		;
		// evtl. wait time if reset of device is necessary and then decide to go to states or ERROR state
		IF (CIf.Job.bolAlmReset = TRUE) THEN
			CIf.Job.eMe_ActivAlmClass := E_AlmClass.NONE; // reset feedback channel for parent
			CIf.Job.bolAlmReset := FALSE;
		END_IF
		// **************************************************************************
		// Wait until Reset all CRC Error is Done
		// **************************************************************************
			fbEcMasterFrameStatisticClearCRC(bExecute:= FALSE);
			// Wait until done
			IF NOT (fbEcMasterFrameStatisticClearCRC.bBusy) THEN
				IF NOT (fbEcMasterFrameStatisticClearCRC.bError) THEN
					bolResetCRCError := FALSE;
				// Error
				ELSE
					// SIf.Alm[E_ALM_ECD.ADS_ComError].strText := 'ADS Communication Error to EtherCAT Master'; // ADS Communication Error to EtherCAT Master => Info = ADS_Errorcode
					pfbAlarmCtrl^.setAlarm(CIf.Info.intCtrlId,E_ALM_ECD.ADS_ComError,UDINT_TO_DINT(fbEcGetSlaveCrcError.nErrId),ADR(SIf.Alm),E_AlmState.RST,CIf.Job.eMe_ActivAlmClass);
					me.StateMachine.intStateNext := cSTA_SUB_ERROR;		
				END_IF
			END_IF
		
		// State Change Condition
		IF ((CIf.Job.bolAlmReset = FALSE) AND (bolResetCRCError = FALSE)) THEN
			IF (me.StateMachine.intStateHistory<=cSTA_PON) THEN
				me.StateMachine.intStateNext := cSTA_PONBusy;
			ELSIF ((SIf.Cfg.bolRunAlways = TRUE) OR (me.intCmd=BASE_PLC.cCMD_RUN)) THEN
				me.StateMachine.intStateNext := cSTA_RUNBusy;
			ELSE
				me.StateMachine.intStateNext := cSTA_OFFBusy;
			END_IF
		END_IF
	END_IF


//--------------------------------------------------------------------------------------
// Exit action
	IF (me.StateMachine.intState<>me.StateMachine.intStateNext) THEN
		;
	END_IF
END_METHOD

METHOD PROTECTED sta_OFF : BOOL
// state implemetation
//--------------------------------------------------------------------------------------
// Entry action
	IF (me.StateMachine.intState<>me.StateMachine.intStateLastCycle) THEN
		me.StateMachine.intStateLastCycle := me.StateMachine.intState;
		// Initialize sub state machine
		me.SubStateMachine.intState:= cSTA_SUB_INITIALIZE; 
		me.SubStateMachine.intStateNext := cSTA_SUB_INITIALIZE;
	END_IF
	
//--------------------------------------------------------------------------------------
// Cyclic action
	IF (me.StateMachine.intState=me.StateMachine.intStateLastCycle) THEN	
		// State Change Condition
		IF (me.Alarm.eActivAlmClass<>E_AlmClass.EOFF) AND (me.Alarm.eActivAlmClass<>E_AlmClass.OFF) THEN	
			IF ((SIf.Cfg.bolRunAlways = TRUE) OR (me.intCmd=BASE_PLC.cCMD_RUN))  THEN
				me.StateMachine.intStateNext := BASE_PLC.cSTA_RUNBusy;
			END_IF
		END_IF
	END_IF

//--------------------------------------------------------------------------------------
// Exit action
	IF (me.StateMachine.intState<>me.StateMachine.intStateNext) THEN
		;
	END_IF
END_METHOD

METHOD PROTECTED sta_PON : BOOL
// state implemetation
//--------------------------------------------------------------------------------------
// Entry action
	IF (me.StateMachine.intState<>me.StateMachine.intStateLastCycle) THEN
		me.StateMachine.intStateLastCycle := me.StateMachine.intState;
		
	END_IF

//--------------------------------------------------------------------------------------
// Cyclic action
	IF (me.StateMachine.intState=me.StateMachine.intStateLastCycle) THEN
		
		;	
		// State Change Condition
		IF ((me.intCmd<>cCMD_PON) AND (me.intCmd<>cCMD_DONE)) OR (SIf.Cfg.bolRunAlways = TRUE) THEN
			me.StateMachine.intStateNext := BASE_PLC.cSTA_OFFBusy;
		END_IF
	END_IF

//--------------------------------------------------------------------------------------
// Exit action
	IF (me.StateMachine.intState<>me.StateMachine.intStateNext) THEN
		;
	END_IF
END_METHOD

METHOD PROTECTED sta_PONBusy : BOOL
VAR
	ii: UINT;
	/// Internal Variable for Found Address
	bolSlaveOK: BOOL;
END_VAR
// state implemetation
//--------------------------------------------------------------------------------------
// Entry action
	IF (me.StateMachine.intState<>me.StateMachine.intStateLastCycle) THEN
		me.StateMachine.intStateLastCycle := me.StateMachine.intState;
		
		udiNumOfStateErrors:= 0;
		udiNumOfCRCErrors:= 0;
		uinLoop:= 0;
		uinSlaveNbr:= 0;

		// Initialize sub state machine
		me.SubStateMachine.intState:= cSTA_SUB_INITIALIZE; 
		me.SubStateMachine.intStateNext := cSTA_SUB_INITIALIZE;
		
		// Get stored alarmtextes into local Texts
		FOR ii := 1 TO (E_ALM_ECD.MAX_E_ALM - 1) DO
			arrAlmtexts[ii] := SIf.Alm[ii].strText;
		END_FOR
	END_IF

//--------------------------------------------------------------------------------------
// Cyclic action
	IF (me.StateMachine.intState=me.StateMachine.intStateLastCycle) THEN
			// Simulation
			IF (CIf.SwCfg.bolSimulation) THEN
				me.SubStateMachine.intStateNext := cSTA_SUB_DONE;
			END_IF
		
			// Sub statemachine to set necessary AMS routes and determine the handle ID of all connections in list	
			CASE me.SubStateMachine.intState OF	
			
				cSTA_SUB_INITIALIZE: 
					me.SubStateMachine.intStateNext := cSTA_SUB_CheckMaster;		

				
				// **************************************************************************
				// Call FUB fbEcGetMasterState to get The State of the EtherCAT Master Device
				// **************************************************************************
				cSTA_SUB_CheckMaster:
				
					// Prepare Function Block
					fbEcGetMasterState(sNetId:= SIf.Cfg.strNetID, 
										bExecute:= FALSE, 
										tTimeout:= UDINT_TO_TIME(SIf.Par.udiTOCheckAll_ms)); 
				
					// Start Function
					fbEcGetMasterState(bExecute:= TRUE, 
										tTimeout:= UDINT_TO_TIME(SIf.Par.udiTOCheckAll_ms)); 
				
					me.SubStateMachine.intStateNext := cSTA_SUB_CheckMasterDone;		
							
				// **************************************************************************
				// Wait until GetAllSlaveAdress is Done
				// **************************************************************************
				cSTA_SUB_CheckMasterDone:
				
					fbEcGetMasterState(bExecute:= FALSE);
					// Wait until done
					IF NOT (fbEcGetMasterState.bBusy) THEN
						IF NOT (fbEcGetMasterState.bError) THEN
							SIf.Cur.worMasterState := fbEcGetMasterState.state;
							// In Operational State check slaves
							IF SIf.Cur.worMasterState = Tc2_EtherCAT.EC_DEVICE_STATE_OP THEN
								me.SubStateMachine.intStateNext := cSTA_SUB_GetAllSlaveAdress;
							// In Pre-Operational check again
							ELSIF ((SIf.Cur.worMasterState = Tc2_EtherCAT.EC_DEVICE_STATE_PREOP) OR (SIf.Cur.worMasterState = Tc2_EtherCAT.EC_DEVICE_STATE_PREOP)) THEN
								me.SubStateMachine.intStateNext := cSTA_SUB_CheckMaster;
							// ELSE ERROR
							ELSE
								// SIf.Alm[E_ALM_ECD.MasterStateError].strText := 'Master State Error'; // Master not in the correct state => Info = Masterstate
								pfbAlarmCtrl^.setAlarm(CIf.Info.intCtrlId,E_ALM_ECD.MasterStateError,WORD_TO_DINT(SIf.Cur.worMasterState),ADR(SIf.Alm),E_AlmState.RST,CIf.Job.eMe_ActivAlmClass);								
							END_IF
						// Error
						ELSE
							// SIf.Alm[E_ALM_ECD.ADS_ComError].strText := 'ADS Communication Error to EtherCAT Master'; // ADS Communication Error to EtherCAT Master => Info = ADS_Errorcode
							pfbAlarmCtrl^.setAlarm(CIf.Info.intCtrlId,E_ALM_ECD.ADS_ComError,UDINT_TO_DINT(fbEcGetMasterState.nErrId),ADR(SIf.Alm),E_AlmState.RST,CIf.Job.eMe_ActivAlmClass);
							me.SubStateMachine.intStateNext := cSTA_SUB_ERROR;		
						END_IF
					END_IF
							
				
				// **************************************************************************
				// Call FUB fbEcGetAllSlaveAddr to get all connected slaves. 
				// **************************************************************************
				cSTA_SUB_GetAllSlaveAdress:
				
					// Prepare Function Block
					fbEcGetAllSlaveAddr(sNetId:= SIf.Cfg.strNetID, 
										pAddrBuf:= ADR(arrSlaveAdress), 
										cbBufLen:= SIZEOF(arrSlaveAdress), 
										bExecute:= FALSE, 
										tTimeout:= UDINT_TO_TIME(SIf.Par.udiTOCheckAll_ms));
				
					// Start Function
					fbEcGetAllSlaveAddr(bExecute:= TRUE, 
										tTimeout:= UDINT_TO_TIME(SIf.Par.udiTOCheckAll_ms));
				
					me.SubStateMachine.intStateNext := cSTA_SUB_GetAllSlaveAdressDone;		
							
				// **************************************************************************
				// Wait until GetAllSlaveAdress is Done
				// **************************************************************************
				cSTA_SUB_GetAllSlaveAdressDone:
				
					fbEcGetAllSlaveAddr(bExecute:= FALSE);
					// Wait until done
					IF NOT (fbEcGetAllSlaveAddr.bBusy) THEN
						IF NOT (fbEcGetAllSlaveAddr.bError) THEN
							// Prepare data
							SIf.Cur.uinNumOfSlaves := fbEcGetAllSlaveAddr.nSlaves;
							IF SIf.Cur.uinNumOfSlaves > 0 THEN
								FOR uinLoop := 0 TO (SIf.Cur.uinNumOfSlaves-1) DO
									SIf.Cur.stSlaveData[uinLoop].uinAddress := arrSlaveAdress[uinLoop];
								END_FOR
							ELSE
								// SIf.Alm[E_ALM_ECD.NoSlaveFound].strText :=  'No Slave in Network'; 		// No EtherCAT Slave found in the network
								pfbAlarmCtrl^.setAlarm(CIf.Info.intCtrlId,E_ALM_ECD.NoSlaveFound,0,ADR(SIf.Alm),E_AlmState.RST,CIf.Job.eMe_ActivAlmClass);								
							END_IF
							me.SubStateMachine.intStateNext := cSTA_SUB_GetConfSlaves;
						// Error
						ELSE
							// SIf.Alm[E_ALM_ECD.ADS_ComError].strText := 'ADS Communication Error to EtherCAT Master'; // ADS Communication Error to EtherCAT Master => Info = ADS_Errorcode
							pfbAlarmCtrl^.setAlarm(CIf.Info.intCtrlId,E_ALM_ECD.ADS_ComError,UDINT_TO_DINT(fbEcGetAllSlaveAddr.nErrId),ADR(SIf.Alm),E_AlmState.RST,CIf.Job.eMe_ActivAlmClass);
							me.SubStateMachine.intStateNext := cSTA_SUB_ERROR;		
						END_IF
					END_IF
			
				// **************************************************************************
				// Call FUB fbEcGetConfSlaves to get all configurated slaves. 
				// **************************************************************************
				cSTA_SUB_GetConfSlaves:
				
					// Prepare Function Block
					fbEcGetConfSlaves(sNetId:= SIf.Cfg.strNetID, 
										pArrEcConfSlaveInfo:= ADR(arrSlaveConf), 
										cbBufLen:= SIZEOF(arrSlaveConf), 
										bExecute:= FALSE, 
										tTimeout:= UDINT_TO_TIME(SIf.Par.udiTOCheckAll_ms));
				
					// Start Function
					fbEcGetConfSlaves(bExecute:= TRUE, 
										tTimeout:= UDINT_TO_TIME(SIf.Par.udiTOCheckAll_ms));
				
					me.SubStateMachine.intStateNext := cSTA_SUB_GetConfSlavesDone;		
							
				// **************************************************************************
				// Wait until fbEcGetConfSlaves is Done
				// **************************************************************************
				cSTA_SUB_GetConfSlavesDone:
				
					fbEcGetConfSlaves(bExecute:= FALSE);
					// Wait until done
					IF NOT (fbEcGetConfSlaves.bBusy) THEN
						IF NOT (fbEcGetConfSlaves.bError) THEN
							// Prepare data
							uinConfigSlaveNbr := fbEcGetConfSlaves.nSlaves;
							IF uinConfigSlaveNbr > 0 THEN
								uinErrorSlaveAdr := 0;
								uinErrorSlaveNbr := 0;
								// Search if configurated Address if found in the hardware found Slaves
								// Loop throug the Configrated Arreay...
								FOR ii := 0 TO (uinConfigSlaveNbr-1) DO	
									bolSlaveOK := FALSE;				
									//...and search in the found addresses	
									FOR uinLoop := 0 TO (SIf.Cur.uinNumOfSlaves-1) DO
										IF (WORD_TO_UINT(arrSlaveConf[ii].nAddr) = SIf.Cur.stSlaveData[uinLoop].uinAddress) THEN // Adress of Configurated and found Slave is the same
											// Copy configuration Data in the CUR Structure
											SIf.Cur.stSlaveData[uinLoop].stConfigData := arrSlaveConf[ii];
											// This slave is done
											bolSlaveOK := TRUE;
											EXIT;
										END_IF
									END_FOR
									// If configurated Address is not found in the redaed Hardware addresses, get Address and increment number
									IF bolSlaveOK = FALSE THEN
										IF uinErrorSlaveAdr = 0 THEN // only write the first module in Error as information
											uinErrorSlaveAdr := WORD_TO_UINT(arrSlaveConf[ii].nAddr);
										END_IF
										uinErrorSlaveNbr := uinErrorSlaveNbr + 1;
									END_IF
								END_FOR
								// Error handling if minimal one configurated slave not found
								IF uinErrorSlaveNbr > 0 THEN 		// Minimal one false Slave
									// Get Error Information
									dinAlarmInfo := UDINT_TO_DINT(SHL(UINT_TO_UDINT(uinErrorSlaveNbr),16) OR uinErrorSlaveAdr);
									strAlarminfo := CONCAT( 'Slave Number: ' , UINT_TO_STRING(uinErrorSlaveAdr));
									strAlarminfo := CONCAT(strAlarminfo, ' of totally missings: ');
									strAlarminfo := CONCAT(strAlarminfo, UDINT_TO_STRING(uinErrorSlaveNbr));
									
									SIf.Alm[E_ALM_ECD.NotAllSlaveConnected].strText := CONCAT(arrAlmtexts[E_ALM_ECD.NotAllSlaveConnected], strAlarminfo);
									
									// SIf.Alm[E_ALM_ECD.NotAllSlaveConnected].strText := 'Configuration and actual differences';// // Configured and reached Slaves are not the same => Info Byte 0+1 = Slave Addres from last error Info Byte 2+3 = Numbers of error Slaves
									pfbAlarmCtrl^.setAlarm(CIf.Info.intCtrlId,E_ALM_ECD.NotAllSlaveConnected,dinAlarmInfo,ADR(SIf.Alm),E_AlmState.RST,CIf.Job.eMe_ActivAlmClass);																	
								END_IF
								// If more slaves hardware found as configurated also an error
								IF SIf.Cur.uinNumOfSlaves > uinConfigSlaveNbr THEN
									// Search if hardware Address which is not configurated
									// Loop throug the Hardware Arreay...
									FOR uinLoop := 0 TO (SIf.Cur.uinNumOfSlaves-1) DO	
										bolSlaveOK := FALSE;				
										//...and search in the configuration
										FOR ii := 0 TO (uinConfigSlaveNbr-1) DO										
											IF (WORD_TO_UINT(arrSlaveConf[ii].nAddr) = SIf.Cur.stSlaveData[uinLoop].uinAddress) THEN // Adress of Configurated and found Slave is the same
												// This slave is done
												bolSlaveOK := TRUE;
												EXIT;
											END_IF
										END_FOR
										// If configurated Address is not found, get Address and increment number
										IF bolSlaveOK = FALSE THEN
											IF uinErrorSlaveAdr = 0 THEN // only write the first module in Error as information
												uinErrorSlaveAdr := WORD_TO_UINT(arrSlaveConf[ii].nAddr);
											END_IF
											uinErrorSlaveNbr := uinErrorSlaveNbr + 1;
										END_IF
									END_FOR
										// Error handling if minimal one configurated slave not found
										IF uinErrorSlaveNbr > 0 THEN 		// Minimal one false Slave
											// Get Error Information
											strAlarminfo := CONCAT(' Slave Number: ' , UINT_TO_STRING(uinErrorSlaveAdr));
											strAlarminfo := CONCAT(strAlarminfo, ' of totally missings: ');
											strAlarminfo := CONCAT(strAlarminfo, UDINT_TO_STRING(uinErrorSlaveNbr));
											
											SIf.Alm[E_ALM_ECD.ToManySlaves].strText := CONCAT(arrAlmtexts[E_ALM_ECD.ToManySlaves], strAlarminfo);
											dinAlarmInfo := UDINT_TO_DINT(SHL(UINT_TO_UDINT(uinErrorSlaveNbr),16) OR uinErrorSlaveAdr);
											// SIf.Alm[E_ALM_ECD.ToManySlaves].strText := 'To many slaves';// More slaves at the master as the structure could handle => Info Byte 0+1 = Slave Addres from last error Info Byte 2+3 = Numbers of error Slaves
											pfbAlarmCtrl^.setAlarm(CIf.Info.intCtrlId,E_ALM_ECD.ToManySlaves,dinAlarmInfo,ADR(SIf.Alm),E_AlmState.RST,CIf.Job.eMe_ActivAlmClass);																	
										END_IF										
								END_IF
							// No Slaves in Cofiguration Found	
							ELSE
								// SIf.Alm[E_ALM_ECD.NoSlaveFound].strText :=  'No Slave in Network'; 		// No EtherCAT Slave found in the network
								pfbAlarmCtrl^.setAlarm(CIf.Info.intCtrlId,E_ALM_ECD.NoSlaveFound,0,ADR(SIf.Alm),E_AlmState.RST,CIf.Job.eMe_ActivAlmClass);								
							END_IF
							me.SubStateMachine.intStateNext := cSTA_SUB_DONE;
						// Error
						ELSE
							// SIf.Alm[E_ALM_ECD.ADS_ComError].strText := 'ADS Communication Error to EtherCAT Master'; // ADS Communication Error to EtherCAT Master => Info = ADS_Errorcode
							pfbAlarmCtrl^.setAlarm(CIf.Info.intCtrlId,E_ALM_ECD.ADS_ComError,UDINT_TO_DINT(fbEcGetConfSlaves.nErrorId),ADR(SIf.Alm),E_AlmState.RST,CIf.Job.eMe_ActivAlmClass);
							me.SubStateMachine.intStateNext := cSTA_SUB_ERROR;		
						END_IF
					END_IF
			

				
				// **************************************************************************
				// All necessary AMS routes set and connection handles are determined 
				// **************************************************************************
				cSTA_SUB_DONE:
				
				// **************************************************************************
				// Error
				// **************************************************************************
				cSTA_SUB_ERROR:
				
			END_CASE	
			
		
		// State Change Condition
		IF ((me.SubStateMachine.intState=cSTA_SUB_ERROR) OR (me.StateMachine.udiTimeInState_ms >= SIf.Par.udiTOPowerOn_ms)) THEN
			// In case if TO
			IF (me.StateMachine.udiTimeInState_ms >= SIf.Par.udiTOPowerOn_ms) THEN
				// SIf.Alm[E_ALM_ECD.TimeOutFunction].strText := 'Timeout EtherCAT function'; // A Function is not finished after the defined Timeout
				pfbAlarmCtrl^.setAlarm(CIf.Info.intCtrlId,E_ALM_ECD.TimeOutFunction,UDINT_TO_DINT(me.StateMachine.udiTimeInState_ms),ADR(SIf.Alm),E_AlmState.RST,CIf.Job.eMe_ActivAlmClass);
			END_IF
			me.StateMachine.intStateNext := cSTA_ERROR;				
		ELSIF (me.SubStateMachine.intState=cSTA_SUB_DONE) THEN
			me.StateMachine.intStateNext := cSTA_PON;
		END_IF
			
	END_IF

//--------------------------------------------------------------------------------------
// Exit action
	IF (me.StateMachine.intState<>me.StateMachine.intStateNext) THEN
		;
	END_IF
END_METHOD

METHOD PROTECTED sta_RUN : BOOL
VAR
	/// internal Loop Variable
	intI: INT;
	/// Internal Variable for Found Address
	bolAlaveOK: BOOL;
END_VAR
// state implemetation
//--------------------------------------------------------------------------------------
// Entry action
	IF (me.StateMachine.intState<>me.StateMachine.intStateLastCycle) THEN
		me.StateMachine.intStateLastCycle := me.StateMachine.intState;
		
		udiNumOfStateErrors:= 0;
		udiNumOfCRCErrors:= 0;
		uinLoop:= 0;
		uinSlaveNbr:= 0;

		// Initialize sub state machine
		me.SubStateMachine.intState:= cSTA_SUB_INITIALIZE; 
		me.SubStateMachine.intStateNext := cSTA_SUB_INITIALIZE;
		
	END_IF

//--------------------------------------------------------------------------------------
// Cyclic action
	IF (me.StateMachine.intState=me.StateMachine.intStateLastCycle) THEN
			// Simulation
			IF (CIf.SwCfg.bolSimulation) THEN
				me.SubStateMachine.intStateNext := cSTA_SUB_WAIT_NEXT_POLL;
				me.SubStateMachine.udiTimeInState_ms := 0;
			END_IF
			
			// Check if a Reset of the CRC Errors has to be done
			IF ((SIf.Alm[E_ALM_ECD.SlaveCRCError].bol = TRUE) AND (CIf.Job.bolAlmReset = TRUE)) THEN
				bolResetCRCError := TRUE;
				SIf.Alm[E_ALM_ECD.SlaveCRCError].bol := FALSE;
			END_IF
			
		
			// Sub statemachine to set necessary AMS routes and determine the handle ID of all connections in list	
			CASE me.SubStateMachine.intState OF	
			
				cSTA_SUB_INITIALIZE: 
					me.SubStateMachine.intStateNext := cSTA_SUB_CheckMaster;		

				
				// **************************************************************************
				// Call FUB fbEcGetMasterState to get The State of the EtherCAT Master Device
				// **************************************************************************
				cSTA_SUB_CheckMaster:
				
					// Prepare Function Block
					fbEcGetMasterState(sNetId:= SIf.Cfg.strNetID, 
										bExecute:= FALSE, 
										tTimeout:= UDINT_TO_TIME(SIf.Par.udiTOCheckAll_ms)); 
				
					// Start Function
					fbEcGetMasterState(bExecute:= TRUE, 
										tTimeout:= UDINT_TO_TIME(SIf.Par.udiTOCheckAll_ms)); 
				
					me.SubStateMachine.intStateNext := cSTA_SUB_CheckMasterDone;		
							
				// **************************************************************************
				// Wait until GetAllSlaveAdress is Done
				// **************************************************************************
				cSTA_SUB_CheckMasterDone:
				
					fbEcGetMasterState(bExecute:= FALSE);
					// Wait until done
					IF NOT (fbEcGetMasterState.bBusy) THEN
						IF NOT (fbEcGetMasterState.bError) THEN
							SIf.Cur.worMasterState := fbEcGetMasterState.state;
							SIf.Cur.worMasterState := fbEcGetMasterState.state;
							// In Operational State check slaves
							IF SIf.Cur.worMasterState = Tc2_EtherCAT.EC_DEVICE_STATE_OP THEN
								me.SubStateMachine.intStateNext := cSTA_SUB_GetAllSlaveAdress;
							// In Pre-Operational check again
							ELSIF ((SIf.Cur.worMasterState = Tc2_EtherCAT.EC_DEVICE_STATE_PREOP) OR (SIf.Cur.worMasterState = Tc2_EtherCAT.EC_DEVICE_STATE_PREOP)) THEN
								me.SubStateMachine.intStateNext := cSTA_SUB_CheckMaster;
							// ELSE ERROR
							ELSE
								// SIf.Alm[E_ALM_ECD.MasterStateError].strText := 'Master State Error'; // Master not in the correct state => Info = Masterstate
								pfbAlarmCtrl^.setAlarm(CIf.Info.intCtrlId,E_ALM_ECD.MasterStateError,WORD_TO_DINT(SIf.Cur.worMasterState),ADR(SIf.Alm),E_AlmState.RST,CIf.Job.eMe_ActivAlmClass);								
							END_IF
						// Error
						ELSE
							// SIf.Alm[E_ALM_ECD.ADS_ComError].strText := 'ADS Communication Error to EtherCAT Master'; // ADS Communication Error to EtherCAT Master => Info = ADS_Errorcode
							pfbAlarmCtrl^.setAlarm(CIf.Info.intCtrlId,E_ALM_ECD.ADS_ComError,UDINT_TO_DINT(fbEcGetMasterState.nErrId),ADR(SIf.Alm),E_AlmState.RST,CIf.Job.eMe_ActivAlmClass);
							me.SubStateMachine.intStateNext := cSTA_SUB_ERROR;		
						END_IF
					END_IF
							
				
				// **************************************************************************
				// Call FUB fbEcGetAllSlaveAddr to get all connected slaves. 
				// **************************************************************************
				cSTA_SUB_GetAllSlaveAdress:
				
					// Prepare Function Block
					fbEcGetAllSlaveAddr(sNetId:= SIf.Cfg.strNetID, 
										pAddrBuf:= ADR(arrSlaveAdress), 
										cbBufLen:= SIZEOF(arrSlaveAdress), 
										bExecute:= FALSE, 
										tTimeout:= UDINT_TO_TIME(SIf.Par.udiTOCheckAll_ms));
				
					// Start Function
					fbEcGetAllSlaveAddr(bExecute:= TRUE, 
										tTimeout:= UDINT_TO_TIME(SIf.Par.udiTOCheckAll_ms));
				
					me.SubStateMachine.intStateNext := cSTA_SUB_GetAllSlaveAdressDone;		
							
				// **************************************************************************
				// Wait until GetAllSlaveAdress is Done
				// **************************************************************************
				cSTA_SUB_GetAllSlaveAdressDone:
				
					fbEcGetAllSlaveAddr(bExecute:= FALSE);
					// Wait until done
					IF NOT (fbEcGetAllSlaveAddr.bBusy) THEN
						IF NOT (fbEcGetAllSlaveAddr.bError) THEN
							// Prepare data
							SIf.Cur.uinNumOfSlaves := fbEcGetAllSlaveAddr.nSlaves;
							IF SIf.Cur.uinNumOfSlaves > 0 THEN
								FOR uinLoop := 0 TO (SIf.Cur.uinNumOfSlaves-1) DO
									SIf.Cur.stSlaveData[uinLoop].uinAddress := arrSlaveAdress[uinLoop];
								END_FOR
							ELSE
								// SIf.Alm[E_ALM_ECD.NoSlaveFound].strText :=  'No Slave in Network'; 		// No EtherCAT Slave found in the network
								pfbAlarmCtrl^.setAlarm(CIf.Info.intCtrlId,E_ALM_ECD.NoSlaveFound,0,ADR(SIf.Alm),E_AlmState.RST,CIf.Job.eMe_ActivAlmClass);								
							END_IF
							me.SubStateMachine.intStateNext := cSTA_SUB_GetConfSlaves;
						// Error
						ELSE
							// SIf.Alm[E_ALM_ECD.ADS_ComError].strText := 'ADS Communication Error to EtherCAT Master'; // ADS Communication Error to EtherCAT Master => Info = ADS_Errorcode
							pfbAlarmCtrl^.setAlarm(CIf.Info.intCtrlId,E_ALM_ECD.ADS_ComError,UDINT_TO_DINT(fbEcGetAllSlaveAddr.nErrId),ADR(SIf.Alm),E_AlmState.RST,CIf.Job.eMe_ActivAlmClass);
							me.SubStateMachine.intStateNext := cSTA_SUB_ERROR;		
						END_IF
					END_IF
			
				// **************************************************************************
				// Call FUB fbEcGetConfSlaves to get all configurated slaves. 
				// **************************************************************************
				cSTA_SUB_GetConfSlaves:
				
					// Prepare Function Block
					fbEcGetConfSlaves(sNetId:= SIf.Cfg.strNetID, 
										pArrEcConfSlaveInfo:= ADR(arrSlaveConf), 
										cbBufLen:= SIZEOF(arrSlaveConf), 
										bExecute:= FALSE, 
										tTimeout:= UDINT_TO_TIME(SIf.Par.udiTOCheckAll_ms));
				
					// Start Function
					fbEcGetConfSlaves(bExecute:= TRUE, 
										tTimeout:= UDINT_TO_TIME(SIf.Par.udiTOCheckAll_ms));
				
					me.SubStateMachine.intStateNext := cSTA_SUB_GetConfSlavesDone;		
							
				// **************************************************************************
				// Wait until fbEcGetConfSlaves is Done
				// **************************************************************************
				cSTA_SUB_GetConfSlavesDone:
				
					fbEcGetConfSlaves(bExecute:= FALSE);
					// Wait until done
					IF NOT (fbEcGetConfSlaves.bBusy) THEN
						IF NOT (fbEcGetConfSlaves.bError) THEN
							// Prepare data
							uinConfigSlaveNbr := fbEcGetConfSlaves.nSlaves;
							IF uinConfigSlaveNbr > 0 THEN
								uinErrorSlaveAdr := 0;
								uinErrorSlaveNbr := 0;
								// Search if configurated Address if found in the hardware found Slaves
								// Loop throug the Configrated Arreay...
								FOR intI := 0 TO (UINT_TO_INT(uinConfigSlaveNbr)-1) DO	
									bolAlaveOK := FALSE;				
									//...and search in the found addresses	
									FOR uinLoop := 0 TO (SIf.Cur.uinNumOfSlaves-1) DO
										IF (WORD_TO_UINT(arrSlaveConf[intI].nAddr) = SIf.Cur.stSlaveData[uinLoop].uinAddress) THEN // Adress of Configurated and found Slave is the same
											// Copy configuration Data in the CUR Structure
											SIf.Cur.stSlaveData[uinLoop].stConfigData := arrSlaveConf[intI];
											// This slave is done
											bolAlaveOK := TRUE;
											EXIT;
										END_IF
									END_FOR
									// If configurated Address is not found in the redaed Hardware addresses, get Address and increment number
									IF bolAlaveOK = FALSE THEN
										IF uinErrorSlaveAdr = 0 THEN // only write the first module in Error as information
											uinErrorSlaveAdr := WORD_TO_UINT(arrSlaveConf[intI].nAddr);
										END_IF
										uinErrorSlaveNbr := uinErrorSlaveNbr + 1;
									END_IF
								END_FOR
								// Error handling if minimal one configurated slave not found
								IF uinErrorSlaveNbr > 0 THEN 		// Minimal one false Slave
									// Get Error Information
									dinAlarmInfo := UDINT_TO_DINT(SHL(UINT_TO_UDINT(uinErrorSlaveNbr),16) OR uinErrorSlaveAdr);
									strAlarminfo := CONCAT(' Slave Number: ' , UINT_TO_STRING(uinErrorSlaveAdr));
									strAlarminfo := CONCAT(strAlarminfo, ' of totally missings: ');
									strAlarminfo := CONCAT(strAlarminfo, UDINT_TO_STRING(uinErrorSlaveNbr));
									SIf.Alm[E_ALM_ECD.NotAllSlaveConnected].strText := CONCAT(arrAlmtexts[E_ALM_ECD.NotAllSlaveConnected], strAlarminfo);
									
									// SIf.Alm[E_ALM_ECD.NotAllSlaveConnected].strText := 'Configuration and actual differences';// // Configured and reached Slaves are not the same => Info Byte 0+1 = Slave Addres from last error Info Byte 2+3 = Numbers of error Slaves
									pfbAlarmCtrl^.setAlarm(CIf.Info.intCtrlId,E_ALM_ECD.NotAllSlaveConnected,dinAlarmInfo,ADR(SIf.Alm),E_AlmState.RST,CIf.Job.eMe_ActivAlmClass);																	
								END_IF
								// If more slaves hardware found as configurated also an error
								IF SIf.Cur.uinNumOfSlaves > uinConfigSlaveNbr THEN
									// Search if hardware Address which is not configurated
									// Loop throug the Hardware Arreay...
									FOR uinLoop := 0 TO (SIf.Cur.uinNumOfSlaves-1) DO	
										bolAlaveOK := FALSE;				
										//...and search in the configuration
										FOR intI := 0 TO (UINT_TO_INT(uinConfigSlaveNbr)-1) DO										
											IF (WORD_TO_UINT(arrSlaveConf[intI].nAddr) = SIf.Cur.stSlaveData[uinLoop].uinAddress) THEN // Adress of Configurated and found Slave is the same
												// This slave is done
												bolAlaveOK := TRUE;
												EXIT;
											END_IF
										END_FOR
										// If configurated Address is not found, get Address and increment number
										IF bolAlaveOK = FALSE THEN
											IF uinErrorSlaveAdr = 0 THEN // only write the first module in Error as information
												uinErrorSlaveAdr := WORD_TO_UINT(arrSlaveConf[intI].nAddr);
											END_IF
											uinErrorSlaveNbr := uinErrorSlaveNbr + 1;
										END_IF
									END_FOR
										// Error handling if minimal one configurated slave not found
										IF uinErrorSlaveNbr > 0 THEN 		// Minimal one false Slave
											// Get Error Information
											dinAlarmInfo := UDINT_TO_DINT(SHL(UINT_TO_UDINT(uinErrorSlaveNbr),16) OR uinErrorSlaveAdr);
											// Get Error Information
											dinAlarmInfo := UDINT_TO_DINT(SHL(UINT_TO_UDINT(uinErrorSlaveNbr),16) OR uinErrorSlaveAdr);
											strAlarminfo := CONCAT(' Slave Number: ' , UINT_TO_STRING(uinErrorSlaveAdr));
											strAlarminfo := CONCAT(strAlarminfo, ' of totally missings: ');
											strAlarminfo := CONCAT(strAlarminfo, UDINT_TO_STRING(uinErrorSlaveNbr));
											SIf.Alm[E_ALM_ECD.ToManySlaves].strText := CONCAT(arrAlmtexts[E_ALM_ECD.ToManySlaves], strAlarminfo);
											// SIf.Alm[E_ALM_ECD.ToManySlaves].strText := 'To many slaves';// More slaves at the master as the structure could handle => Info Byte 0+1 = Slave Addres from last error Info Byte 2+3 = Numbers of error Slaves
											pfbAlarmCtrl^.setAlarm(CIf.Info.intCtrlId,E_ALM_ECD.ToManySlaves,dinAlarmInfo,ADR(SIf.Alm),E_AlmState.RST,CIf.Job.eMe_ActivAlmClass);																	
										END_IF										
								END_IF
							// No Slaves in Cofiguration Found	
							ELSE
								// SIf.Alm[E_ALM_ECD.NoSlaveFound].strText :=  'No Slave in Network'; 		// No EtherCAT Slave found in the network
								pfbAlarmCtrl^.setAlarm(CIf.Info.intCtrlId,E_ALM_ECD.NoSlaveFound,0,ADR(SIf.Alm),E_AlmState.RST,CIf.Job.eMe_ActivAlmClass);								
							END_IF
							me.SubStateMachine.intStateNext := cSTA_SUB_CheckSlaveChanges;
						// Error
						ELSE
							// SIf.Alm[E_ALM_ECD.ADS_ComError].strText := 'ADS Communication Error to EtherCAT Master'; // ADS Communication Error to EtherCAT Master => Info = ADS_Errorcode
							pfbAlarmCtrl^.setAlarm(CIf.Info.intCtrlId,E_ALM_ECD.ADS_ComError,UDINT_TO_DINT(fbEcGetConfSlaves.nErrorId),ADR(SIf.Alm),E_AlmState.RST,CIf.Job.eMe_ActivAlmClass);
							me.SubStateMachine.intStateNext := cSTA_SUB_ERROR;		
						END_IF
					END_IF
					
				// **************************************************************************
				// Call FUB fbEcGetAllSlaveAbnormalStateChanges to get The StateChanges
				// **************************************************************************
				cSTA_SUB_CheckSlaveChanges:
				
					// Prepare Function Block
					fbEcGetAllSlaveAbnormalStateChanges(sNetId:= SIf.Cfg.strNetID, 
										pAddrBuf:= ADR(arrSlaveAbnormalStates), 
										cbBufLen:= SIZEOF(arrSlaveAbnormalStates), 
										bExecute:= FALSE, 
										tTimeout:= UDINT_TO_TIME(SIf.Par.udiTOCheckAll_ms)); 
				
					// Start Function
					fbEcGetAllSlaveAbnormalStateChanges(bExecute:= TRUE, 
										tTimeout:= UDINT_TO_TIME(SIf.Par.udiTOCheckAll_ms)); 
				
					me.SubStateMachine.intStateNext := cSTA_SUB_CheckSlaveChangesDone;		
							
				// **************************************************************************
				// Wait until GetAllSlaveAdress is Done
				// **************************************************************************
				cSTA_SUB_CheckSlaveChangesDone:
				
					fbEcGetAllSlaveAbnormalStateChanges(bExecute:= FALSE);
					// Wait until done
					IF NOT (fbEcGetAllSlaveAbnormalStateChanges.bBusy) THEN
						IF NOT (fbEcGetAllSlaveAbnormalStateChanges.bError) THEN
							// Check Data
							uinErrorSlaveAdr := 0;
							uinErrorSlaveNbr := 0;
							uinErrorSlaveInfo := 0;
							FOR uinLoop := 0 TO (SIf.Cur.uinNumOfSlaves-1) DO
								IF arrSlaveAbnormalStates[uinLoop] > 0 THEN
									IF uinErrorSlaveAdr = 0 THEN // only write the first module in Error as information
										uinErrorSlaveAdr := uinLoop;
										uinErrorSlaveInfo := UDINT_TO_UINT(arrSlaveAbnormalStates[uinLoop]);
									END_IF
									uinErrorSlaveNbr := uinErrorSlaveNbr + 1;
								END_IF
							END_FOR
							// Error from a Slave with too many State Changes
							IF uinErrorSlaveNbr > 0 THEN
								// Get Error Information
								dinAlarmInfo := UDINT_TO_DINT(SHL(UINT_TO_UDINT(uinErrorSlaveNbr),16) OR uinErrorSlaveAdr);
								strAlarminfo := CONCAT(' Slave Number: ' , UINT_TO_STRING(uinErrorSlaveAdr));
								strAlarminfo := CONCAT(strAlarminfo, ' with Errors: ');
								strAlarminfo := CONCAT(strAlarminfo, UDINT_TO_STRING(uinErrorSlaveInfo));
								SIf.Alm[E_ALM_ECD.StateChanges].strText := CONCAT(arrAlmtexts[E_ALM_ECD.StateChanges], strAlarminfo);
								// SIf.Alm[E_ALM_ECD.SlaveCRCError].strText :=  'Slave CRC Error';	// Minimum one Slave has to many CRC Erros => Byte 0+1 = Slave Addres from last error, Info Byte 2 + 3 = Number of CRC Errors from last Slave with error
								pfbAlarmCtrl^.setAlarm(CIf.Info.intCtrlId,E_ALM_ECD.StateChanges,dinAlarmInfo,ADR(SIf.Alm),E_AlmState.RST,CIf.Job.eMe_ActivAlmClass);																								
							END_IF
							me.SubStateMachine.intStateNext := cSTA_SUB_SLAVE_START;
						// Error
						ELSE
							// SIf.Alm[E_ALM_ECD.ADS_ComError].strText := 'ADS Communication Error to EtherCAT Master'; // ADS Communication Error to EtherCAT Master => Info = ADS_Errorcode
							pfbAlarmCtrl^.setAlarm(CIf.Info.intCtrlId,E_ALM_ECD.ADS_ComError,UDINT_TO_DINT(fbEcGetAllSlaveAbnormalStateChanges.nErrId),ADR(SIf.Alm),E_AlmState.RST,CIf.Job.eMe_ActivAlmClass);
							me.SubStateMachine.intStateNext := cSTA_SUB_ERROR;		
						END_IF
					END_IF
							
				
				
				// **************************************************************************
				// Prepare Data for Slave Checks 
				// **************************************************************************
				cSTA_SUB_SLAVE_START:
					uinLoopSlave := 0;
					uinErrorSlaveAdr := 0;
					uinErrorSlaveNbr := 0;
					uinErrorSlaveInfo := 0;
					uinErrorSlaveAdrCRC := 0;
					uinErrorSlaveNbrCRC := 0;
					uinErrorSlaveInfoCRC := 0;
					uinErrorSlaveLink := 0;
					uinErrorSlaveLinkNbr := 0;
					uinErrorSlaveLinkInfo := 0;
					me.SubStateMachine.intStateNext := cSTA_SUB_CheckSlaveState;
					
				// **************************************************************************
				// Call FUB fbEcGetSlaveState to get the State of 
				// **************************************************************************
				cSTA_SUB_CheckSlaveState:
				
					// Prepare Function Block
					fbEcGetSlaveState(sNetId:= SIf.Cfg.strNetID, 
										nSlaveAddr:= SIf.Cur.stSlaveData[uinLoopSlave].uinAddress, 
										bExecute:= FALSE, 
										tTimeout:= UDINT_TO_TIME(SIf.Par.udiTOCheckOne_ms));
				
					// Start Function
					fbEcGetSlaveState(bExecute:= TRUE, 
										nSlaveAddr:= SIf.Cur.stSlaveData[uinLoopSlave].uinAddress, 
										tTimeout:= UDINT_TO_TIME(SIf.Par.udiTOCheckOne_ms));
				
					me.SubStateMachine.intStateNext := cSTA_SUB_CheckSlaveStateDone;		
							
				// **************************************************************************
				// Wait until GetAllSlaveAdress is Done
				// **************************************************************************
				cSTA_SUB_CheckSlaveStateDone:
				
					fbEcGetSlaveState(bExecute:= FALSE);
					// Wait until done
					IF NOT (fbEcGetSlaveState.bBusy) THEN
						IF NOT (fbEcGetSlaveState.bError) THEN
							// Check State of Slave
							SIf.Cur.stSlaveData[uinLoopSlave].stState := fbEcGetSlaveState.state;
							IF (SIf.Cur.stSlaveData[uinLoopSlave].stState.deviceState <> Tc2_EtherCAT.EC_DEVICE_STATE_OP) THEN
								IF uinErrorSlaveAdr = 0 THEN // only write the first module in Error as information
									uinErrorSlaveAdr := SIf.Cur.stSlaveData[uinLoopSlave].uinAddress;
									uinErrorSlaveInfo := SIf.Cur.stSlaveData[uinLoopSlave].stState.deviceState;
								END_IF
								uinErrorSlaveNbr := uinErrorSlaveNbr+1;
							END_IF
							// Check Link State
							// Word 1 = State, Word 2 = Port
							IF ((SIf.Cur.stSlaveData[uinLoopSlave].stState.linkState AND 16#0F) > 0) THEN
								IF uinErrorSlaveLink = 0 THEN // only write the first module in Error as information
									uinErrorSlaveLink := SIf.Cur.stSlaveData[uinLoopSlave].uinAddress;
									uinErrorSlaveLinkInfo := SIf.Cur.stSlaveData[uinLoopSlave].stState.linkState;
								END_IF
								uinErrorSlaveLinkNbr := uinErrorSlaveNbr+1;
							END_IF
							me.SubStateMachine.intStateNext := cSTA_SUB_CheckCRC;
						// Error
						ELSE
							// SIf.Alm[E_ALM_ECD.ADS_ComError].strText := 'ADS Communication Error to EtherCAT Master'; // ADS Communication Error to EtherCAT Master => Info = ADS_Errorcode
							pfbAlarmCtrl^.setAlarm(CIf.Info.intCtrlId,E_ALM_ECD.ADS_ComError,UDINT_TO_DINT(fbEcGetSlaveState.nErrId),ADR(SIf.Alm),E_AlmState.RST,CIf.Job.eMe_ActivAlmClass);
							me.SubStateMachine.intStateNext := cSTA_SUB_ERROR;		
						END_IF
					END_IF
			
				// **************************************************************************
				// Call FUB fbEcGetSlaveCrcError to get the CRC Errors of the Slaves
				// **************************************************************************
				cSTA_SUB_CheckCRC:
				
					// Prepare Function Block
					fbEcGetSlaveCrcError(sNetId:= SIf.Cfg.strNetID, 
										nSlaveAddr:= SIf.Cur.stSlaveData[uinLoopSlave].uinAddress, 
										bExecute:= FALSE, 
										tTimeout:= UDINT_TO_TIME(SIf.Par.udiTOCheckOne_ms));
				
					// Start Function
					fbEcGetSlaveCrcError(bExecute:= TRUE, 
										nSlaveAddr:= SIf.Cur.stSlaveData[uinLoopSlave].uinAddress, 
										tTimeout:= UDINT_TO_TIME(SIf.Par.udiTOCheckOne_ms));
				
					me.SubStateMachine.intStateNext := cSTA_SUB_CheckCRCDone;		
							
				// **************************************************************************
				// Wait until GetAllSlaveAdress is Done
				// **************************************************************************
				cSTA_SUB_CheckCRCDone:
				
					fbEcGetSlaveCrcError(bExecute:= FALSE);
					// Wait until done
					IF NOT (fbEcGetSlaveCrcError.bBusy) THEN
						IF NOT (fbEcGetSlaveCrcError.bError) THEN
							// Check data
							SIf.Cur.stSlaveData[uinLoopSlave].stCRCError := fbEcGetSlaveCrcError.crcError;
							IF (SIf.Cur.stSlaveData[uinLoopSlave].stCRCError.portA >= SIf.Par.udiMaxCRC) THEN
								IF ( (uinErrorSlaveAdrCRC = 0) OR (uinErrorSlaveInfoCRC < UDINT_TO_UINT(SIf.Cur.stSlaveData[uinLoopSlave].stCRCError.portA)) ) THEN // only write the first module in Error as information or the slave with the most CRC errors
									uinErrorSlaveAdrCRC := SIf.Cur.stSlaveData[uinLoopSlave].uinAddress;
									uinErrorSlaveInfoCRC := UDINT_TO_UINT(SIf.Cur.stSlaveData[uinLoopSlave].stCRCError.portA);
								END_IF
								uinErrorSlaveNbrCRC := uinErrorSlaveNbrCRC + 1;
							END_IF
							IF (SIf.Cur.stSlaveData[uinLoopSlave].stCRCError.portB >= SIf.Par.udiMaxCRC) THEN
								IF ( (uinErrorSlaveAdrCRC = 0) OR (uinErrorSlaveInfoCRC < UDINT_TO_UINT(SIf.Cur.stSlaveData[uinLoopSlave].stCRCError.portA)) ) THEN // only write the first module in Error as information or the slave with the most CRC errors
									uinErrorSlaveAdrCRC := SIf.Cur.stSlaveData[uinLoopSlave].uinAddress;
									uinErrorSlaveInfoCRC := UDINT_TO_UINT(SIf.Cur.stSlaveData[uinLoopSlave].stCRCError.portB);
								END_IF
								uinErrorSlaveNbrCRC := uinErrorSlaveNbrCRC + 1;
							END_IF
							IF (SIf.Cur.stSlaveData[uinLoopSlave].stCRCError.portC >= SIf.Par.udiMaxCRC) THEN
								IF ( (uinErrorSlaveAdrCRC = 0) OR (uinErrorSlaveInfoCRC < UDINT_TO_UINT(SIf.Cur.stSlaveData[uinLoopSlave].stCRCError.portA)) ) THEN // only write the first module in Error as information or the slave with the most CRC errors
									uinErrorSlaveAdrCRC := SIf.Cur.stSlaveData[uinLoopSlave].uinAddress;
									uinErrorSlaveInfoCRC := UDINT_TO_UINT(SIf.Cur.stSlaveData[uinLoopSlave].stCRCError.portC);
								END_IF
								uinErrorSlaveNbrCRC := uinErrorSlaveNbrCRC + 1;
							END_IF
							IF (SIf.Cur.stSlaveData[uinLoopSlave].stCRCError.portD >= SIf.Par.udiMaxCRC) THEN
								IF ( (uinErrorSlaveAdrCRC = 0) OR (uinErrorSlaveInfoCRC < UDINT_TO_UINT(SIf.Cur.stSlaveData[uinLoopSlave].stCRCError.portA)) ) THEN // only write the first module in Error as information or the slave with the most CRC errors
									uinErrorSlaveAdrCRC := SIf.Cur.stSlaveData[uinLoopSlave].uinAddress;
									uinErrorSlaveInfoCRC := UDINT_TO_UINT(SIf.Cur.stSlaveData[uinLoopSlave].stCRCError.portD);
								END_IF
								uinErrorSlaveNbrCRC := uinErrorSlaveNbrCRC + 1;
							END_IF
							me.SubStateMachine.intStateNext := cSTA_SUB_Inc;
						// Error
						ELSE
							// SIf.Alm[E_ALM_ECD.ADS_ComError].strText := 'ADS Communication Error to EtherCAT Master'; // ADS Communication Error to EtherCAT Master => Info = ADS_Errorcode
							pfbAlarmCtrl^.setAlarm(CIf.Info.intCtrlId,E_ALM_ECD.ADS_ComError,UDINT_TO_DINT(fbEcGetSlaveCrcError.nErrId),ADR(SIf.Alm),E_AlmState.RST,CIf.Job.eMe_ActivAlmClass);
							me.SubStateMachine.intStateNext := cSTA_SUB_ERROR;		
						END_IF
					END_IF

				//************************************************************************
				// Prepare Function for next Slave 
				//************************************************************************	
				cSTA_SUB_Inc:
					IF (uinLoopSlave < (SIf.Cur.uinNumOfSlaves-1)) THEN
						// Another slave to check
						uinLoopSlave := uinLoopSlave + 1;
						me.SubStateMachine.intStateNext := cSTA_SUB_CheckSlaveState;
					// Otherwise all slaves are checked
					ELSE
						// Check states
						// Error handling if minimal one configurated slave not found
						IF uinErrorSlaveNbr > 0 THEN 		// Minimal one false Slave
							// Get Error Information
							dinAlarmInfo := UDINT_TO_DINT(SHL(UINT_TO_UDINT(uinErrorSlaveInfo),16) OR uinErrorSlaveAdr);
							strAlarminfo := CONCAT(' Slave Number: ' , UINT_TO_STRING(uinErrorSlaveAdr));
							strAlarminfo := CONCAT(strAlarminfo, ' in State: ');
							strAlarminfo := CONCAT(strAlarminfo, UDINT_TO_STRING(uinErrorSlaveInfo));
							SIf.Alm[E_ALM_ECD.SlaveStateError].strText := CONCAT(arrAlmtexts[E_ALM_ECD.SlaveStateError], strAlarminfo);
							// SIf.Alm[E_ALM_ECD.SlaveStateError].strText := 'Slave State Error'; // Minimum one Slave not in the correct state => Byte 0+1 = Slave Addres from last error, Info Byte 2 + 3 = State of last error Slave
							pfbAlarmCtrl^.setAlarm(CIf.Info.intCtrlId,E_ALM_ECD.SlaveStateError,dinAlarmInfo,ADR(SIf.Alm),E_AlmState.RST,CIf.Job.eMe_ActivAlmClass);																	
						END_IF	
						// Check Link Error
						IF uinErrorSlaveLinkNbr > 0 THEN 		// Minimal one false Slave
							// Get Error Information
							dinAlarmInfo := UDINT_TO_DINT(SHL(UINT_TO_UDINT(uinErrorSlaveLinkInfo),16) OR uinErrorSlaveLink);
							strAlarminfo := CONCAT(' Slave Number:  ' , UINT_TO_STRING(uinErrorSlaveLink));
							strAlarminfo := CONCAT(strAlarminfo, ' Link Error: ');
							strAlarminfo := CONCAT(strAlarminfo, UDINT_TO_STRING(uinErrorSlaveLinkInfo));
							SIf.Alm[E_ALM_ECD.SlaveLinkError].strText := CONCAT(arrAlmtexts[E_ALM_ECD.SlaveLinkError], strAlarminfo);
							// SIf.Alm[E_ALM_ECD.SlaveLinkError].strText :=  'Slave Link State Error'; // Minimum one Slave has a LinkState Erros => Byte 0+1 = Slave Addres from last error Info Byte 2 + 3 = Link State of last error Slave
							pfbAlarmCtrl^.setAlarm(CIf.Info.intCtrlId,E_ALM_ECD.SlaveLinkError,dinAlarmInfo,ADR(SIf.Alm),E_AlmState.RST,CIf.Job.eMe_ActivAlmClass);																	
						END_IF	
						// Check CRC Errors
						SIf.Cur.udiCRCSumm := 0;
						FOR uinLoop := 0 TO (SIf.Cur.uinNumOfSlaves-1) DO
							// Add all CRC Errors for informations   
							SIf.Cur.udiCRCSumm := SIf.Cur.udiCRCSumm + SIf.Cur.stSlaveData[uinLoop].stCRCError.portA + SIf.Cur.stSlaveData[uinLoop].stCRCError.portB + SIf.Cur.stSlaveData[uinLoop].stCRCError.portC + SIf.Cur.stSlaveData[uinLoop].stCRCError.portD;
						END_FOR
						// Error from a Slave with too many CRC Errors
						IF uinErrorSlaveNbrCRC > 0 THEN
							// Get Error Information
							dinAlarmInfo := UDINT_TO_DINT(SHL(UINT_TO_UDINT(uinErrorSlaveInfoCRC),16) OR uinErrorSlaveAdrCRC);
							strAlarminfo := CONCAT(' Slave Number: ' , UINT_TO_STRING(uinErrorSlaveAdrCRC));
							strAlarminfo := CONCAT(strAlarminfo, ' CRC Errors: ');
							strAlarminfo := CONCAT(strAlarminfo, UDINT_TO_STRING(uinErrorSlaveInfoCRC));
							SIf.Alm[E_ALM_ECD.SlaveCRCError].strText := CONCAT(arrAlmtexts[E_ALM_ECD.SlaveCRCError], strAlarminfo);
							// SIf.Alm[E_ALM_ECD.SlaveCRCError].strText :=  'Slave CRC Error';	// Minimum one Slave has to many CRC Erros => Byte 0+1 = Slave Addres from last error, Info Byte 2 + 3 = Number of CRC Errors from last Slave with error
							pfbAlarmCtrl^.setAlarm(CIf.Info.intCtrlId,E_ALM_ECD.SlaveCRCError,dinAlarmInfo,ADR(SIf.Alm),E_AlmState.RST,CIf.Job.eMe_ActivAlmClass);																								
							SIf.Alm[E_ALM_ECD.SlaveCRCError].bol := TRUE;
						END_IF
						me.SubStateMachine.intStateNext := cSTA_SUB_WAIT_NEXT_POLL;
						
					END_IF
		
				//************************************************************************
				// Wait for next polling - Connection list completely processed 
				//************************************************************************	
				cSTA_SUB_WAIT_NEXT_POLL:
				
					// Wait polling time expired 	
					IF (me.SubStateMachine.udiTimeInState_ms >= SIf.Par.udiPollingInterval_ms) THEN				
						//Start again at first connection in list
						me.SubStateMachine.intStateNext := cSTA_SUB_INITIALIZE;
					ELSIF bolResetCRCError = TRUE THEN
						me.SubStateMachine.intStateNext := cSTA_SUB_CheckCRCReset;						
					END_IF
					
				// **************************************************************************
				// Call FUB fbEcMasterFrameStatisticClearCRC to reset all CRC Errors of the Slaves
				// **************************************************************************
				cSTA_SUB_CheckCRCReset:
				
					// Prepare Function Block
					fbEcMasterFrameStatisticClearCRC(sNetId:= SIf.Cfg.strNetID, 
										bExecute:= FALSE, 
										tTimeout:= UDINT_TO_TIME(SIf.Par.udiTOCheckAll_ms));
				
					// Start Function
					fbEcMasterFrameStatisticClearCRC(bExecute:= TRUE, 
										tTimeout:= UDINT_TO_TIME(SIf.Par.udiTOCheckAll_ms));
				
					me.SubStateMachine.intStateNext := cSTA_SUB_CheckCRCResetDone;		
							
				// **************************************************************************
				// Wait until Reset all CRC Error is Done
				// **************************************************************************
				cSTA_SUB_CheckCRCResetDone:
				
					fbEcMasterFrameStatisticClearCRC(bExecute:= FALSE);
					// Wait until done
					IF NOT (fbEcMasterFrameStatisticClearCRC.bBusy) THEN
						IF NOT (fbEcMasterFrameStatisticClearCRC.bError) THEN
							me.SubStateMachine.intStateNext := cSTA_SUB_WAIT_NEXT_POLL;
							bolResetCRCError := FALSE;
						// Error
						ELSE
							// SIf.Alm[E_ALM_ECD.ADS_ComError].strText := 'ADS Communication Error to EtherCAT Master'; // ADS Communication Error to EtherCAT Master => Info = ADS_Errorcode
							pfbAlarmCtrl^.setAlarm(CIf.Info.intCtrlId,E_ALM_ECD.ADS_ComError,UDINT_TO_DINT(fbEcGetSlaveCrcError.nErrId),ADR(SIf.Alm),E_AlmState.RST,CIf.Job.eMe_ActivAlmClass);
							me.SubStateMachine.intStateNext := cSTA_SUB_ERROR;		
						END_IF
					END_IF

				//************************************************************************
				// ERROR			
				//************************************************************************	
				cSTA_SUB_ERROR:
					// SIf.Alm[E_ALM_ECD.ADS_ComError].strText := 'ADS Communication Error to EtherCAT Master'; // ADS Communication Error to EtherCAT Master => Info = ADS_Errorcode
					pfbAlarmCtrl^.setAlarm(CIf.Info.intCtrlId,E_ALM_ECD.ADS_ComError,UDINT_TO_DINT(udiFBerror),ADR(SIf.Alm),E_AlmState.RST,CIf.Job.eMe_ActivAlmClass);
					me.StateMachine.intStateNext := BASE_PLC.cSTA_ERROR;	
			
				
			END_CASE	
			
		
		// State Change Condition
		IF ((me.SubStateMachine.intState=cSTA_SUB_ERROR) OR ((me.SubStateMachine.udiTimeInState_ms >= SIf.Par.udiTOPowerOn_ms) AND (me.SubStateMachine.intState <> cSTA_SUB_WAIT_NEXT_POLL))) THEN
			// In case if TO
			IF (me.SubStateMachine.udiTimeInState_ms >= SIf.Par.udiTOPowerOn_ms) THEN
				// SIf.Alm[E_ALM_ECD.TimeOutFunction].strText := 'Timeout EtherCAT function'; // A Function is not finished after the defined Timeout
				pfbAlarmCtrl^.setAlarm(CIf.Info.intCtrlId,E_ALM_ECD.TimeOutFunction,UDINT_TO_DINT(me.SubStateMachine.udiTimeInState_ms),ADR(SIf.Alm),E_AlmState.RST,CIf.Job.eMe_ActivAlmClass);
			END_IF
			me.StateMachine.intStateNext := cSTA_ERROR;				
		END_IF
			
	END_IF

//--------------------------------------------------------------------------------------
// Exit action
	IF (me.StateMachine.intState<>me.StateMachine.intStateNext) THEN
		;
	END_IF
END_METHOD

METHOD PROTECTED sta_RUNBusy : BOOL
// state implemetation
//--------------------------------------------------------------------------------------
// Entry action
	IF (me.StateMachine.intState<>me.StateMachine.intStateLastCycle) THEN
		me.StateMachine.intStateLastCycle := me.StateMachine.intState;
		;
	END_IF

//--------------------------------------------------------------------------------------
// Cyclic action
	IF (me.StateMachine.intState=me.StateMachine.intStateLastCycle) THEN
		IF (TRUE) THEN
			me.StateMachine.intStateNext := BASE_PLC.cSTA_RUN;
		END_IF
	END_IF

//--------------------------------------------------------------------------------------
// Exit action
	IF (me.StateMachine.intState<>me.StateMachine.intStateNext) THEN
		;
	END_IF
END_METHOD

METHOD PROTECTED StateMachine : BOOL
SUPER^.StateMachine();

// main statemachine of base controller
CASE me.StateMachine.intState OF
	cSTA_RUNBusy: 
        THIS^.sta_RUNBusy();
    cSTA_RUN: 
        THIS^.sta_RUN();				
END_CASE;
END_METHOD

END_FUNCTION_BLOCK

// POUs/Controller/Lvl0/RFW (RFID Reader-Writer)/FB_DtChnToLine_NewRFID
FUNCTION_BLOCK FB_DtChnToLine_NewRFID
VAR_INPUT
	bolResetError: BOOL;
	pSIf: POINTER TO T_Ctrl_SIf_RFW;
END_VAR
VAR_OUTPUT
	///Error value
	intError: INT;
END_VAR
VAR
	/// Internal Variable
	intStatemachine: INT;
	/// Time Variables
	fbGetSystemTime: GETSYSTEMTIME;
	stfileTime: T_FILETIME;
	dtActualTime: DT;
	/// Data not correct
	bolDataBad: BOOL;
	/// Retry Counts for error message
	intCountRetry: INT;
	/// Buffer for Senddata
	aBuffer: ARRAY[0..cDtChnBuffer] OF T_NewRFID_DtChn;
	/// Pointer for new Input
	intPBufferInput: INT;
	/// Pointer for readout
	intPBufferOutput: INT;
	/// Data Channel Specific Variable
	intIndexOldest: INT;
	/// Date and time of the oldes imput
	dtOldestTag: DT;
END_VAR
VAR CONSTANT
	cDtChnBuffer: INT := 20;
	cSTA_SUB_Data_Init: INT := 900;
	cSTA_SUB_Data_WaitForJob: INT := 902;
	cSTA_SUB_Data_SendData: INT := 904;
	cSTA_SUB_Data_Acknowledge: INT := 906;
	cSTA_SUB_Data_Retry: INT := 908;
	cSTA_SUB_Data_Error: INT := 910;
	cDataState_DONE: INT := -1;
	cDataState_Ready: INT := 1;
	cDataState_Retry: INT := -99;
	cDataState_Error: INT := -100;
	cMAX_RETRY: INT := 10;
	/// Error Codes
	cERR_BufferFull: INT := -99;
	cERR_NoSIF: INT := -100;
END_VAR

(*__________________________________________________________________________________________________
¦	
¦	Vistaprint Schweiz GmbH
¦	CH - 8401 Winterthur
¦
¦	www.vistaprint.ch - info@vistaprint.ch
¦___________________________________________________________________________________________________

Function desription:
Datachannel to send data to Lince Controller
Insert new Job with Method Creat in a Buffer
Send buffer elements if Linecontroller is ready


History:
Version		Date			Author		Comment
---------------------------------------------------------------------------------------------------
0.00.1		26.08.2013		AVM/PRE		Start history
0.00.2		30.09.2013		AVM/PRE		Date and time with string, not with DT Type

___________________________________________________________________________________________________*)

// Data Channel to Receive Data from Line Controller
// Startup check States
IF (pSIf <> 0) THEN
	IF (intStatemachine < cSTA_SUB_Data_Init) THEN
		intStatemachine := cSTA_SUB_Data_Init;
	END_IF
ELSE
	intError := cERR_NoSIF;
END_IF

CASE intStatemachine OF
	cSTA_SUB_Data_Init:
		IF pSIf^.DtChnToLine.stNewRfid.intDataState = cDataState_DONE THEN
			intStatemachine := cSTA_SUB_Data_WaitForJob;
		END_IF
		
	cSTA_SUB_Data_WaitForJob:
		// New data arrived
		IF intPBufferInput <> intPBufferOutput THEN
			IF pSIf^.DtChnToLine.stNewRfid.intDataState = cDataState_DONE THEN
				intStatemachine := cSTA_SUB_Data_SendData;
			END_IF
		END_IF
	
	cSTA_SUB_Data_SendData:	
		pSIf^.DtChnToLine.stNewRfid.uliTagID := aBuffer[intPBufferOutput].uliTagID;
		pSIf^.DtChnToLine.stNewRfid.strID := aBuffer[intPBufferOutput].strID;
		pSIf^.DtChnToLine.stNewRfid.strTimestamp := aBuffer[intPBufferOutput].strTimestamp;
		pSIf^.DtChnToLine.stNewRfid.intDataState := cDataState_Ready;
		intStatemachine := cSTA_SUB_Data_Acknowledge;	
		
	cSTA_SUB_Data_Acknowledge:	
		IF pSIf^.DtChnToLine.stNewRfid.intDataState = cDataState_DONE THEN
			// Data read from Line Controller
			// Reset Buffer Element
			aBuffer[intPBufferOutput].strTimestamp := '';
			aBuffer[intPBufferOutput].intDataState := 0;
			aBuffer[intPBufferOutput].uliTagID := 0;
			aBuffer[intPBufferOutput].strID := '';
			// Increase Read out pointer
			IF intPBufferOutput < cDtChnBuffer THEN
				intPBufferOutput := intPBufferOutput + 1;
			ELSE
				intPBufferOutput := 0;
			END_IF
			intStatemachine := cSTA_SUB_Data_WaitForJob;
			
		ELSIF pSIf^.DtChnToLine.stNewRfid.intDataState = cDataState_Retry THEN
			intStatemachine := cSTA_SUB_Data_Retry;
		ELSIF pSIf^.DtChnToLine.stNewRfid.intDataState = cDataState_Error THEN
			intStatemachine := cSTA_SUB_Data_Error;
		END_IF
		
	cSTA_SUB_Data_Retry:
			IF intCountRetry < cMAX_RETRY THEN
				intCountRetry := intCountRetry + 1;
				intStatemachine := cSTA_SUB_Data_SendData;
			ELSE
				intStatemachine := cSTA_SUB_Data_Error;
			END_IF

	cSTA_SUB_Data_Error:
		intError := intCountRetry;
		IF bolResetError = TRUE THEN
			intStatemachine := cSTA_SUB_Data_WaitForJob;
		END_IF
			
END_CASE

METHOD Creat : INT
VAR_INPUT
	/// configurable if Tag or Tray ID
	In_strID: STRING;
	In_uliTagID: ULINT;
END_VAR

VAR
	strTemp : STRING;
END_VAR
// Insert a new Job to send at Line controller
// Only insert the job, if the buffer is not full, next input dosn't cross input and Outputpointer

// Get Systemtime
fbGetSystemTime(timeLoDW=>stfileTime.dwLowDateTime, timeHiDW=>stfileTime.dwHighDateTime);
dtActualTime := FILETIME_TO_DT( stfileTime );

IF ((intPBufferInput + 1) = intPBufferOutput) OR ((intPBufferInput = cDtChnBuffer) AND (intPBufferOutput = 0)) THEN
	Creat := cERR_BufferFull;
ELSE
	aBuffer[intPBufferInput].uliTagID := In_uliTagID;
	aBuffer[intPBufferInput].strID := In_strID;
	strTemp := DT_TO_STRING(dtActualTime);
	strTemp := Tc2_Standard.RIGHT(STR:=strTemp, SIZE:= (LEN(strTemp)-3));
	strTemp := CONCAT(strTemp,'.000');	
	aBuffer[intPBufferInput].strTimestamp := strTemp;
	IF intPBufferInput < cDtChnBuffer THEN
		intPBufferInput := intPBufferInput + 1;
	ELSE
		intPBufferInput := 0;
	END_IF
	Creat := intPBufferInput;
END_IF
END_METHOD

END_FUNCTION_BLOCK

// POUs/Controller/Lvl0/RFW (RFID Reader-Writer)/FB_RFW
FUNCTION_BLOCK FB_RFW EXTENDS FB_CtrlBase
VAR_INPUT
	pRFD_SIf: POINTER TO T_RFD;
END_VAR
VAR
	/// Specific interface struct for public access
	SIf: T_Ctrl_SIf_RFW;
	/// Internal Variable
	bolNewTag: BOOL;
	/// Rising Edge New tag at antenna
	bolRENewTag: BOOL;
	/// Read All is finished
	bolAllFinished: BOOL;
	/// Internal Job for more reading
	dwoJobIntern: DWORD;
	/// Startadress on the Tag from the needed Data
	uinDataAdress: UINT;
	/// Lengh of data to read or write
	uinDataLengh: UINT;
	/// old Tag ID to know a new RFID Tag is on antenna
	uliTagID_old: ULINT;
	/// Temporary Help Variable
	usiTemp: USINT;
	/// Temporary Help Variable
	uinTemp: UINT;
	/// Temporary Help Variable
	intTemp: INT;
	intValue: INT;
	/// Temporary Help Variable
	udiTemp: UDINT;
	/// Temporary Help Variable
	uliTemp: LWORD;
	/// Temporary Help Variable
	strTemp: STRING;
	/// Temporary Help Variable to save to position of the point in the string
	intPositionPoint: INT;
	/// Temporary Help Variable to save to position of the - in the string
	intPositionSign: INT;
	/// Short Brake between the different Reads
	udiTimeDelayRead : UDINT;
	/// Data Channel to Line new RFID Tag
	fbDtChnToLine_NewRFID: FB_DtChnToLine_NewRFID;
	intDtChnToLineState: INT;

END_VAR
VAR CONSTANT
	///sub States for RUN Function
	cRFW_SUB_WaitTag: INT := 302;
	cRFW_SUB_SendJob: INT := 304;
	cRFW_SUB_GetData: INT := 306;
	cRFW_SUB_CheckData: INT := 308;
	cRFW_SUB_SendJobTrayID: INT := 310;
	cRFW_SUB_GetDataTrayID: INT := 312;
	cRFW_SUB_CheckDataTrayID: INT := 314;
	cRFW_SUB_Finished: INT := 320;
END_VAR

(*__________________________________________________________________________________________________
¦	
¦	Vistaprint Schweiz GmbH
¦	CH - 8401 Winterthur
¦
¦	www.vistaprint.ch - info@vistaprint.ch
¦___________________________________________________________________________________________________

Function desription:
RFID Reader and Writer
Controlls the communication to the RFID Reader and Writer


History:
Version		Date			Author		Comment
---------------------------------------------------------------------------------------------------
0.00.1		09.07.2013		AVME/PRE	Start history
0.00.2		19.09.2013		AVME/PRE	Implement new Base Concept
0.00.3		24.09.2013		AVME/KVO	Parameter init from element controller to driver
0.00.4		01.10.2013		AVME/PRE	Insert DataChanel to Line
0.00.5		14.11.2013		AVME/PRE	First Checks on the promo machine
0.00.6		17.02.2014		AVME/KVO	Bug fix write single data
___________________________________________________________________________________________________*)


SUPER^();

(*
IF (me.bolActivate) THEN // cyclic call enabled
	IF (CIf.Info.bolInitDone=FALSE) THEN // first cycle -> init
		CtrlInit();
		CIf.Info.bolInitDone := TRUE;
	ELSE
		CycleStartDuty();
	
		Always();
		
		StateMachine();
		
		CycleEndDuty();
	END_IF
END_IF;
*)

METHOD PROTECTED Always : BOOL
SUPER^.Always();

// ----------------------------------------------------------------------------------
// cyclic actions outside of statemachine
IF (me.StateMachine.intState<>cSTA_SINGLE_ANSWER) THEN
	pRFD_SIf^.stCur.pData := ADR(SIf.Cur.abytData[0]);
	SIf.Cur.bolPresent := pRFD_SIf^.stStatus.bolPresent;
	IF (CIf.Job.bolAlmReset = TRUE) AND (pRFD_SIf^.stErr.bolErrorActive = TRUE) THEN
		pRFD_SIf^.stErr.bolErrAck := TRUE;
	END_IF
	
	// Data channel to UI/Line
	fbDtChnToLine_NewRFID.pSIf := ADR(SIf);
	fbDtChnToLine_NewRFID.bolResetError := CIf.Job.bolAlmReset;
	fbDtChnToLine_NewRFID();
	IF fbDtChnToLine_NewRFID.intError <> 0 THEN
		// Set Alarm: SIf.Alm[6].strText := 'Data Channel Error Send Data';
		//pfbAlarmCtrl^.setAlarm(CIf.Info.intCtrlId,6,fbDtChnToLine_NewRFID.intError,ADR(SIf.Alm),E_AlmState.RST,CIf.Job.eMe_ActivAlmClass);	
	END_IF
	
	// config driver
	pRFD_SIf^.stCfg.bolSimulation := CIf.SwCfg.bolSimulation;
	pRFD_SIf^.stCfg.eTyp := SIf.Cfg.eTyp;
	pRFD_SIf^.stCfg.stNetId := SIf.Cfg.stNetId; //PLC NetId
	pRFD_SIf^.stCfg.uinSlaveAddr := SIf.Cfg.uinSlaveAddr; //Io card Ethercat adress 
	
	// ----------------------------------------------------------------------------------
	// Always change actions in Base Library
	// ----------------------------------------------------------------------------------
	// overrule error always from base -> no EOFF State!! in EOFF go to OFF
	IF (me.StateMachine.intStateNext = cSTA_EOFFBusy) THEN
		IF (me.StateMachine.intState=cSTA_OFF) THEN
			me.StateMachine.intStateNext := cSTA_OFF;
		ELSE // stay in OFF
			me.StateMachine.intStateNext := cSTA_OFFBusy;
		END_IF
	END_IF
END_IF
END_METHOD

METHOD FB_init : BOOL
VAR_INPUT
	///if TRUE, the retain variables are initialized (warm start / cold start)
	bInitRetains: BOOL;
	///if TRUE, the instance afterwards gets moved into the copy code (online change)
	bInCopyCode: BOOL;
END_VAR
VAR
	udiTaskCnt: UDINT;
	ii: UINT;
END_VAR
//------------------------------------------------------------------------------------------------------------------------
// to manually change in new FUB implementation!!!
// define valid commands for this controller
FOR ii:= 0 TO (SIZEOF(CIf.Job.aCmdList)/SIZEOF(CIf.Job.aCmdList[0])-1) BY 1 DO
	IF (CIf.Job.aCmdList[ii].intCmd=cCMD_INITIALIZED) THEN
		// found first empty array element
		EXIT;
	END_IF
END_FOR
CIf.Job.aCmdList[ii].intCmd := RFW_CmdState.cCMD_READ;
CIf.Job.aCmdList[ii].strName := 'Read'; 
CIf.Job.aCmdList[ii].bolAvailable := TRUE;
ii := ii +1;
CIf.Job.aCmdList[ii].intCmd := RFW_CmdState.cCMD_WRITE;
CIf.Job.aCmdList[ii].strName := 'Write';
CIf.Job.aCmdList[ii].bolAvailable := TRUE;
ii := ii +1;
CIf.Job.aCmdList[ii].intCmd := RFW_CmdState.cCMD_ON;
CIf.Job.aCmdList[ii].strName := 'On';
CIf.Job.aCmdList[ii].bolAvailable := TRUE;
ii := ii +1;
CIf.Job.aCmdList[ii].intCmd := cCMD_RUN;
CIf.Job.aCmdList[ii].strName := 'Run';
CIf.Job.aCmdList[ii].bolAvailable := TRUE;

// set name of class/typ
CIf.Info.strType := 'FB_RFID';
CIf.Info.strFullName := 'RFID Reader-Writer';

// set alarm class
SIf.Alm[1].eAlmClass := E_AlmClass.TSTOP;
SIf.Alm[1].strText := 'Communication Error between PLC and RFID Reader'; 
SIf.Alm[2].eAlmClass := E_AlmClass.TSTOP;
SIf.Alm[2].strText := 'Initialisation Error from RFID Reader';
SIf.Alm[3].eAlmClass := E_AlmClass.TSTOP;
SIf.Alm[3].strText := 'RFID Tag Error';
SIf.Alm[4].eAlmClass := E_AlmClass.TSTOP;
SIf.Alm[4].strText := 'timeout wait on Data';
SIf.Alm[5].eAlmClass := E_AlmClass.TSTOP;
SIf.Alm[5].strText := 'Command for this type of RFID not possible';
SIf.Alm[6].eAlmClass := E_AlmClass.INFO;
SIf.Alm[6].strText := 'Data Channel Error Send Data';

//*******************************************************************************
// initial values
//*******************************************************************************

// software configuration
CIf.SwCfg.bolExist := TRUE;
CIf.SwCfg.bolSimulation := FALSE;

// parmeter
SIf.Par.udiReadTime_ms := 30000;
SIf.Par.udiWriteTime_ms := 300000;
SIf.Par.udiMinCmdTime := 100;

// Get correct type
SIf.Cfg.eTyp := E_Typ_RFW.RF382R;
SIf.Cfg.stNetId := '192.168.2.123.1.1'; //PLC NetId
SIf.Cfg.uinSlaveAddr := 1039; //Io card Ethercat adress 
SIf.Cfg.bolGetTrayIDAuto := FALSE;
SIf.Cfg.bolDtChToLine_send := TRUE;
END_METHOD

METHOD PROTECTED getCmdState : STRING
VAR_INPUT
	intCmdState: INT;
	bolState: BOOL;
END_VAR
getCmdState := SUPER^.getCmdState(intCmdState:=intCmdState,bolState:=bolState); // get global/base defined cmds/states
IF (getCmdState='') THEN // global not defined get local
	// get string cmd/state string information in runtime
	IF (bolState=FALSE) THEN
		// cmd's
		CASE intCmdState OF
			RFW_CmdState.cCMD_ON: 
				getCmdState := 'cCMD_ON';
			RFW_CmdState.cCMD_READ: 
				getCmdState := 'cCMD_READ';
			RFW_CmdState.cCMD_WRITE: 
				getCmdState := 'cCMD_WRITE';
		END_CASE;
	ELSE
	
	// cmd's
		CASE intCmdState OF
			RFW_CmdState.cSTA_ONBusy: 
				getCmdState := 'cSTA_ONBusy';
			RFW_CmdState.cSTA_ON: 
				getCmdState := 'cSTA_ON';
			RFW_CmdState.cSTA_READBusy: 
				getCmdState := 'cSTA_READBusy';
			RFW_CmdState.cSTA_READ: 
				getCmdState := 'cSTA_READ';
			RFW_CmdState.cSTA_WRITEBusy: 
				getCmdState := 'cSTA_WRITEBusy';
			RFW_CmdState.cSTA_WRITE: 
				getCmdState := 'cSTA_WRITE';
				
			// SUB States
			cRFW_SUB_WaitTag:
				getCmdState := 'cRFW_SUB_WaitTag';
			cRFW_SUB_SendJob:
				getCmdState := 'cRFW_SUB_SendJob';
			cRFW_SUB_GetData:
				getCmdState := 'cRFW_SUB_GetData';
			cRFW_SUB_CheckData:
				getCmdState := 'cRFW_SUB_CheckData';
			cRFW_SUB_SendJobTrayID:
				getCmdState := 'cRFW_SUB_SendJobTrayID';
			cRFW_SUB_GetDataTrayID:
				getCmdState := 'cRFW_SUB_GetDataTrayID';
			cRFW_SUB_CheckDataTrayID:
				getCmdState := 'cRFW_SUB_CheckDataTrayID';
			cRFW_SUB_Finished: 			
				getCmdState := 'cRFW_SUB_Finished';
		END_CASE;
	END_IF
END_IF
END_METHOD

METHOD getCtrlSIf : POINTER TO T_Ctrl_SIf_RFW
getCtrlSIf := ADR(SIf);
END_METHOD

METHOD PROTECTED IoInBridge : BOOL
// digitale and analoge inputs read from hardware or forcing

IF (CIf.SwCfg.bolSimulation = FALSE) THEN
	;
	//ctrl.In.bol_PosSwitchBasicDefTyp.intern := getInBol(ctrl.ifc.Job.bol_Force ,ADR(ctrl.In.bol_PosSwitchBasicDefTyp);
ELSE
	//simulation of global IO
END_IF
END_METHOD

METHOD PROTECTED IoOutBridge : BOOL
VAR
	bolSwitchValvesOff: BOOL;
END_VAR
// digitale and analoge inputs read from hardware or forcing
IF (CIf.SwCfg.bolSimulation = FALSE) THEN
	// check interlocks to prevent damages
	IF (CIf.Job.bolIlkOverwrite=FALSE) THEN
		;
	END_IF
END_IF
END_METHOD

METHOD PROTECTED sta_ERROR : BOOL
// state implemetation
//--------------------------------------------------------------------------------------
// Entry action
	IF (me.StateMachine.intState<>me.StateMachine.intStateLastCycle) THEN
		me.StateMachine.intStateHistory := me.StateMachine.intStateLastCycle; // -> possibillity to go back to state before error
		me.StateMachine.intStateLastCycle := me.StateMachine.intState;
	END_IF


//--------------------------------------------------------------------------------------
// Cyclic action
	IF (me.StateMachine.intState=me.StateMachine.intStateLastCycle) THEN
		
		IF (pRFD_SIf^.stErr.bolComError = TRUE) OR (pRFD_SIf^.stErr.bolProtcolError = TRUE) THEN
			// SIf.Alm[1].strText := 'Communication Error between PLC and RFID Reader'; 
			pfbAlarmCtrl^.setAlarm(CIf.Info.intCtrlId,1,UDINT_TO_DINT(pRFD_SIf^.stErr.udiErrorID),ADR(SIf.Alm),E_AlmState.RST,CIf.Job.eMe_ActivAlmClass);
		ELSIF pRFD_SIf^.stErr.bolSDOError = TRUE THEN
			// SIf.Alm[2].strText := 'Initialisation Error from RFID Reader';
			pfbAlarmCtrl^.setAlarm(CIf.Info.intCtrlId,2,UDINT_TO_DINT(pRFD_SIf^.stErr.udiErrorID),ADR(SIf.Alm),E_AlmState.RST,CIf.Job.eMe_ActivAlmClass);
		ELSIF (pRFD_SIf^.stErr.bolRFIDError = TRUE) THEN
			// SIf.Alm[3].strText := 'RFID Tag Error';
			pfbAlarmCtrl^.setAlarm(CIf.Info.intCtrlId,3,UDINT_TO_DINT(pRFD_SIf^.stErr.udiErrorID),ADR(SIf.Alm),E_AlmState.RST,CIf.Job.eMe_ActivAlmClass);
		END_IF
		
		
		// State Change Condition
		IF (CIf.Job.bolAlmReset = TRUE) THEN
			me.StateMachine.intStateNext := cSTA_ERRORQuit;
		END_IF
	END_IF




//--------------------------------------------------------------------------------------
// Exit action
	IF (me.StateMachine.intState<>me.StateMachine.intStateNext) THEN
		IF 	CIf.Job.intACmd > cCMD_OFF THEN
			CIf.Job.intACmd := cCMD_DONE;
		END_IF

	END_IF
END_METHOD

METHOD PROTECTED sta_OFF : BOOL
// state implemetation
//--------------------------------------------------------------------------------------
// Entry action
	IF (me.StateMachine.intState<>me.StateMachine.intStateLastCycle) THEN
		me.StateMachine.intStateLastCycle := me.StateMachine.intState;
		
	END_IF


//--------------------------------------------------------------------------------------
// Cyclic action
	IF (me.StateMachine.intState=me.StateMachine.intStateLastCycle) THEN
		
		;
		
		
		// State Change Condition
		IF (me.Alarm.eActivAlmClass<>E_AlmClass.EOFF) AND (me.Alarm.eActivAlmClass<>E_AlmClass.OFF) THEN
			IF(me.intCmd=cCMD_RUN) THEN
				me.StateMachine.intStateNext := cSTA_RUNBusy;
			ELSIF ((me.intCmd=RFW_CmdState.cCMD_READ) OR (me.intCmd=RFW_CmdState.cCMD_WRITE)) AND (SIf.Cfg.eTyp = E_Typ_RFW.RF382R) THEN
				// SIf.Alm[5].strText := 'Command for this type of RFID not possible';
				pfbAlarmCtrl^.setAlarm(CIf.Info.intCtrlId,5,UDINT_TO_DINT(pRFD_SIf^.stErr.udiErrorID),ADR(SIf.Alm),E_AlmState.RST,CIf.Job.eMe_ActivAlmClass);			
			ELSIF(me.intCmd=RFW_CmdState.cCMD_READ) THEN
				me.StateMachine.intStateNext := RFW_CmdState.cSTA_READBusy;
			ELSIF(me.intCmd=RFW_CmdState.cCMD_WRITE) THEN
				me.StateMachine.intStateNext := RFW_CmdState.cSTA_WRITEBusy;
			ELSIF(me.intCmd=RFW_CmdState.cCMD_ON) THEN
				me.StateMachine.intStateNext := RFW_CmdState.cSTA_ONBusy;			
			END_IF
		END_IF
	END_IF




//--------------------------------------------------------------------------------------
// Exit action
	IF (me.StateMachine.intState<>me.StateMachine.intStateNext) THEN
		;
	END_IF
END_METHOD

METHOD PROTECTED sta_OFFBusy : BOOL
// state implemetation
//--------------------------------------------------------------------------------------
// Entry action
	IF (me.StateMachine.intState<>me.StateMachine.intStateLastCycle) THEN
		me.StateMachine.intStateLastCycle := me.StateMachine.intState;
		fbSimulationTimer.IN := FALSE;
		fbSimulationTimer.PT := UDINT_TO_TIME(SIf.Par.udiReadTime_ms / 2);
		fbSimulationTimer(); // set time/reset timer
		fbSimulationTimer.IN := TRUE; // start timer
		
	END_IF


//--------------------------------------------------------------------------------------
// Cyclic action
	IF (me.StateMachine.intState=me.StateMachine.intStateLastCycle) THEN
		// Simulation
		IF (CIf.SwCfg.bolSimulation) THEN
			fbSimulationTimer(); // simulation time
			IF (fbSimulationTimer.Q) THEN
				pRFD_SIf^.intCmd := RFD_Cmd.cRFD_CMD_DONE;
				SIf.Cur.bolPresent := FALSE;
			END_IF
		END_IF
		
	
		// State Change Condition
		IF pRFD_SIf^.stErr.bolErrorActive = TRUE THEN // AND (me.StateMachine.udiTimeInState_ms>SIf.Par.udiWriteTime_ms) 
			me.StateMachine.intStateNext :=  cSTA_ERROR;
		//ELSIF(pRFD_SIf^.intCmd = RFD_Cmd.cRFD_CMD_DONE) THEN
		ELSIF (TRUE) THEN
			me.StateMachine.intStateNext := cSTA_OFF;
		END_IF
	END_IF




//--------------------------------------------------------------------------------------
// Exit action
	IF (me.StateMachine.intState<>me.StateMachine.intStateNext) THEN
		;
	END_IF
END_METHOD

METHOD PROTECTED sta_ON : BOOL
// state implemetation
//--------------------------------------------------------------------------------------
// Entry action
	IF (me.StateMachine.intState<>me.StateMachine.intStateLastCycle) THEN
		me.StateMachine.intStateLastCycle := me.StateMachine.intState;
		bolNewTag := FALSE;
		me.SubStateMachine.intState := cRFW_SUB_WaitTag-1; // init first state - string
		me.SubStateMachine.intStateNext := cRFW_SUB_WaitTag;
		fbSimulationTimer.IN := FALSE;
		fbSimulationTimer.PT := UDINT_TO_TIME(SIf.Par.udiReadTime_ms / 2);
		fbSimulationTimer(); // set time/reset timer
		fbSimulationTimer.IN := TRUE; // start timer
		
	END_IF


//--------------------------------------------------------------------------------------
// Cyclic action
	IF (me.StateMachine.intState=me.StateMachine.intStateLastCycle) THEN

		// Simulation
		
		// Function
				
		// State Change Condition
		IF (pRFD_SIf^.stErr.bolErrorActive = TRUE) THEN  
			me.StateMachine.intStateNext :=  cSTA_ERROR;
		ELSIF ((me.intCmd=cCMD_READ) OR (me.intCmd=cCMD_WRITE)) AND (SIf.Cfg.eTyp = E_Typ_RFW.RF382R) THEN
			// SIf.Alm[5].strText := 'Command for this type of RFID not possible';
			pfbAlarmCtrl^.setAlarm(CIf.Info.intCtrlId,5,UDINT_TO_DINT(pRFD_SIf^.stErr.udiErrorID),ADR(SIf.Alm),E_AlmState.RST,CIf.Job.eMe_ActivAlmClass);			
		ELSIF (me.intCmd=cCMD_READ) THEN
			me.StateMachine.intStateNext := cSTA_READBusy;
		ELSIF(me.intCmd=cCMD_WRITE) THEN
			me.StateMachine.intStateNext := cSTA_WRITEBusy;
		ELSIF(me.intCmd=cCMD_RUN) THEN
			me.StateMachine.intStateNext := cSTA_RUNBusy;			
		END_IF
	END_IF




//--------------------------------------------------------------------------------------
// Exit action
	IF (me.StateMachine.intState<>me.StateMachine.intStateNext) THEN
		;		
	END_IF
END_METHOD

METHOD PROTECTED sta_ONbusy : BOOL
// state implemetation
//--------------------------------------------------------------------------------------
// Entry action
	IF (me.StateMachine.intState<>me.StateMachine.intStateLastCycle) THEN
		me.StateMachine.intStateLastCycle := me.StateMachine.intState;
		bolNewTag := FALSE;
		me.SubStateMachine.intState := cRFW_SUB_WaitTag;
		
		fbSimulationTimer.IN := FALSE;
		fbSimulationTimer.PT := UDINT_TO_TIME(SIf.Par.udiReadTime_ms / 2);
		fbSimulationTimer(); // set time/reset timer
		fbSimulationTimer.IN := TRUE; // start timer
		
	END_IF


//--------------------------------------------------------------------------------------
// Cyclic action
	IF (me.StateMachine.intState=me.StateMachine.intStateLastCycle) THEN

		// Simulation
		IF (CIf.SwCfg.bolSimulation) THEN
			pRFD_SIf^.stStatus.bolOn := TRUE;
			fbSimulationTimer(); // simulation time
			IF (fbSimulationTimer.Q) THEN
				;
			END_IF
		END_IF
		
		// Function
		IF(pRFD_SIf^.stStatus.bolOn = FALSE) THEN
			pRFD_SIf^.intCmd := RFD_Cmd.cRFD_CMD_CTRL_ON;
		END_IF
		
		// State Change Condition
		IF (pRFD_SIf^.stErr.bolErrorActive = TRUE) THEN  
			me.StateMachine.intStateNext :=  cSTA_ERROR;
		ELSIF(pRFD_SIf^.stStatus.bolOn = TRUE) THEN
			me.StateMachine.intStateNext := RFW_CmdState.cSTA_ON;
		END_IF
	END_IF




//--------------------------------------------------------------------------------------
// Exit action
	IF (me.StateMachine.intState<>me.StateMachine.intStateNext) THEN
		;		
	END_IF
END_METHOD

METHOD PROTECTED sta_PON : BOOL
// state implemetation
//--------------------------------------------------------------------------------------
// Entry action
	IF (me.StateMachine.intState<>me.StateMachine.intStateLastCycle) THEN
		me.StateMachine.intStateLastCycle := me.StateMachine.intState;
		
	END_IF


//--------------------------------------------------------------------------------------
// Cyclic action
	IF (me.StateMachine.intState=me.StateMachine.intStateLastCycle) THEN
		
		;
		
		
		// State Change Condition
		IF (me.intCmd<>cCMD_PON) AND (me.intCmd<>cCMD_DONE) THEN
			me.StateMachine.intStateNext := cSTA_OFFBusy;
		END_IF
	END_IF




//--------------------------------------------------------------------------------------
// Exit action
	IF (me.StateMachine.intState<>me.StateMachine.intStateNext) THEN
		;
	END_IF
END_METHOD

METHOD PROTECTED sta_PONBusy : BOOL
// state implemetation
//--------------------------------------------------------------------------------------
// Entry action
	IF (me.StateMachine.intState<>me.StateMachine.intStateLastCycle) THEN
		me.StateMachine.intStateLastCycle := me.StateMachine.intState;
		fbSimulationTimer.IN := FALSE;
		fbSimulationTimer.PT := UDINT_TO_TIME(SIf.Par.udiReadTime_ms / 2);
		fbSimulationTimer(); // set time/reset timer
		fbSimulationTimer.IN := TRUE; // start timer
		
		IF (CIf.SwCfg.bolSimulation = FALSE) THEN
			pRFD_SIf^.intCmd := RFD_Cmd.cRFD_CMD_CTRL_ON; // parameter initialisation on driver
		END_IF
	END_IF


//--------------------------------------------------------------------------------------
// Cyclic action
	IF (me.StateMachine.intState=me.StateMachine.intStateLastCycle) THEN
		// Simulation
		IF (CIf.SwCfg.bolSimulation) THEN
			fbSimulationTimer(); // simulation time
			IF (fbSimulationTimer.Q) THEN
				pRFD_SIf^.intCmd := RFD_Cmd.cRFD_CMD_DONE;
				SIf.Cur.bolPresent := FALSE;
			END_IF
		END_IF
		
	
		// State Change Condition
		IF (pRFD_SIf^.stErr.bolErrorActive = TRUE) AND (CIf.SwCfg.bolSimulation = FALSE) THEN // AND (me.StateMachine.udiTimeInState_ms>SIf.Par.udiWriteTime_ms) 
			me.StateMachine.intStateNext :=  cSTA_ERROR;
		ELSIF (pRFD_SIf^.intCmd = RFD_Cmd.cRFD_CMD_DONE) THEN
			me.StateMachine.intStateNext := cSTA_PON;
		END_IF
	END_IF




//--------------------------------------------------------------------------------------
// Exit action
	IF (me.StateMachine.intState<>me.StateMachine.intStateNext) THEN
		;
	END_IF
END_METHOD

METHOD PROTECTED sta_READ : BOOL
// state implemetation
//--------------------------------------------------------------------------------------
// Entry action
	IF (me.StateMachine.intState<>me.StateMachine.intStateLastCycle) THEN
		me.StateMachine.intStateLastCycle := me.StateMachine.intState;

	END_IF


//--------------------------------------------------------------------------------------
// Cyclic action
	IF (me.StateMachine.intState=me.StateMachine.intStateLastCycle) THEN

		// Simulation
		IF (CIf.SwCfg.bolSimulation) THEN
			;
		END_IF
		
		// State Change Condition
		IF(me.intCmd=cCMD_RUN) THEN
			me.StateMachine.intStateNext := cSTA_RUNBusy;
		ELSIF ((me.intCmd=RFW_CmdState.cCMD_READ) OR (me.intCmd=RFW_CmdState.cCMD_WRITE)) AND (SIf.Cfg.eTyp = E_Typ_RFW.RF382R) THEN
			// SIf.Alm[5].strText := 'Command for this type of RFID not possible';
			pfbAlarmCtrl^.setAlarm(CIf.Info.intCtrlId,5,UDINT_TO_DINT(pRFD_SIf^.stErr.udiErrorID),ADR(SIf.Alm),E_AlmState.RST,CIf.Job.eMe_ActivAlmClass);			
		ELSIF(me.intCmd=RFW_CmdState.cCMD_WRITE) THEN
			me.StateMachine.intStateNext := RFW_CmdState.cSTA_WRITEBusy;
		//ELSIF(me.intCmd=RFW_CmdState.cCMD_READ) THEN
		//	me.StateMachine.intStateNext := RFW_CmdState.cSTA_READBusy;
		ELSIF(me.intCmd=RFW_CmdState.cCMD_ON) THEN
			me.StateMachine.intStateNext := RFW_CmdState.cSTA_ONBusy;			
		END_IF
	END_IF




//--------------------------------------------------------------------------------------
// Exit action
	IF (me.StateMachine.intState<>me.StateMachine.intStateNext) THEN
		;
	END_IF
END_METHOD

METHOD PROTECTED sta_READBusy : BOOL
// state implemetation
//--------------------------------------------------------------------------------------
// Entry action
	IF (me.StateMachine.intState<>me.StateMachine.intStateLastCycle) THEN
		me.StateMachine.intStateLastCycle := me.StateMachine.intState;
		
		fbSimulationTimer.IN := FALSE;
		fbSimulationTimer.PT := UDINT_TO_TIME(SIf.Par.udiReadTime_ms / 2);
		fbSimulationTimer(); // set time/reset timer
		fbSimulationTimer.IN := TRUE; // start timer
		
		IF SIf.Cur.dwoJob = 0 THEN
			SIf.Cur.dwoJob := RFID_Data.cRFID_AllData;
		END_IF
		
		bolAllFinished := FALSE;
		dwoJobIntern := SIf.Cur.dwoJob;
		
		uinDataAdress := DWORD_TO_UINT(dwoJobIntern);
		uinDataAdress := uinDataAdress MOD 16#100;							// Maximum 255 data
		
		pRFD_SIf^.stCur.uinAdressData := uinDataAdress;
		pRFD_SIf^.stCur.uinAdressTag := DWORD_TO_UINT(dwoJobIntern);
		pRFD_SIf^.stCur.usiCount := DWORD_TO_USINT(SHR(dwoJobIntern,16));
		
		udiTimeDelayRead := 0;

		IF (CIf.SwCfg.bolSimulation = FALSE) THEN
			pRFD_SIf^.intCmd := RFD_Cmd.cRFD_CMD_Read;
		END_IF
	END_IF


//--------------------------------------------------------------------------------------
// Cyclic action
	IF (me.StateMachine.intState=me.StateMachine.intStateLastCycle) THEN

		// Simulation
		IF (CIf.SwCfg.bolSimulation) THEN
			fbSimulationTimer(); // simulation time
			IF (fbSimulationTimer.Q) THEN
				pRFD_SIf^.intCmd := RFD_Cmd.cRFD_CMD_DONE;
			END_IF
		END_IF
		
		// Function
		// By Read all the Tray ID has to be readed too
		IF (pRFD_SIf^.intCmd = RFD_Cmd.cRFD_CMD_DONE) AND (udiTimeDelayRead > SIf.Par.udiMinCmdTime) THEN
		//---------------------------------------
			udiTimeDelayRead := 0;
			// Prepare Data from read memory
			// Repetition ID
			IF (dwoJobIntern = RFID_Data.cRFID_AllData) OR (dwoJobIntern = RFID_Data.cRFID_RepetionID) THEN
				uinDataAdress := DWORD_TO_UINT(RFID_Data.cRFID_RepetionID);
				uinDataAdress := uinDataAdress  MOD 16#100;							// only 0..255
				IF ((uinDataAdress >= 0) AND (uinDataAdress <= 255)) THEN
					SIf.Cur.stData.usiRepetitionID := SIf.Cur.abytData[uinDataAdress];
				END_IF
			END_IF
			// Tray Info
			IF (dwoJobIntern = RFID_Data.cRFID_AllData) OR (dwoJobIntern = RFID_Data.cRFID_TrayInfo) THEN
				uinDataAdress := DWORD_TO_UINT(RFID_Data.cRFID_TrayInfo);
				uinDataAdress := uinDataAdress  MOD 16#100;							// only 0..255
				IF ((uinDataAdress >= 0) AND (uinDataAdress <= 255)) THEN
					SIf.Cur.stData.bolWorkstation2 := SIf.Cur.abytData[uinDataAdress].0;
					SIf.Cur.stData.bolDeleteFileAfterPrint := SIf.Cur.abytData[uinDataAdress].6;
					SIf.Cur.stData.bolPrintOk := SIf.Cur.abytData[uinDataAdress].7;
				END_IF
			END_IF
			// Height of tray
			IF (dwoJobIntern = RFID_Data.cRFID_AllData) OR (dwoJobIntern = RFID_Data.cRFID_HeighOfTray) THEN
				uinDataAdress := DWORD_TO_UINT(RFID_Data.cRFID_HeighOfTray);
				uinDataAdress := uinDataAdress  MOD 16#100;							// only 0..255
				IF ((uinDataAdress >= 0) AND (uinDataAdress <= 255)) THEN
					SIf.Cur.stData.bolHeightUseMeasure := SIf.Cur.abytData[uinDataAdress].0;
					SIf.Cur.stData.usiHeightOffset := 0;
					SIf.Cur.stData.usiHeightOffset.0 := SIf.Cur.abytData[uinDataAdress].1;
					SIf.Cur.stData.usiHeightOffset.1 := SIf.Cur.abytData[uinDataAdress].2;
					SIf.Cur.stData.usiHeightOffset.2 := SIf.Cur.abytData[uinDataAdress].3;
					SIf.Cur.stData.bolHeightOffsetSignMinus := SIf.Cur.abytData[uinDataAdress].4;
				END_IF
			END_IF
			// Pretreatment
			IF (dwoJobIntern = RFID_Data.cRFID_AllData) OR (dwoJobIntern = RFID_Data.cRFID_RepetionID) THEN
				uinDataAdress := DWORD_TO_UINT(RFID_Data.cRFID_Pretreatment);
				uinDataAdress := uinDataAdress  MOD 16#100;							// only 0..255
				IF ((uinDataAdress >= 0) AND (uinDataAdress <= 255)) THEN
					SIf.Cur.stData.bolIonizer := SIf.Cur.abytData[uinDataAdress].1;
					SIf.Cur.stData.usiPlasmaLevel := 0;
					SIf.Cur.stData.usiPlasmaLevel.0 := SIf.Cur.abytData[uinDataAdress].2;
					SIf.Cur.stData.usiPlasmaLevel.1 := SIf.Cur.abytData[uinDataAdress].3;
					SIf.Cur.stData.bolPrintPass := SIf.Cur.abytData[uinDataAdress].4;
					SIf.Cur.stData.bolNozzleCheck := SIf.Cur.abytData[uinDataAdress].5;
					SIf.Cur.stData.bolAligneCheck := SIf.Cur.abytData[uinDataAdress].6;
				END_IF
			END_IF
			// UV-curing
			IF (dwoJobIntern = RFID_Data.cRFID_AllData) OR (dwoJobIntern = RFID_Data.cRFID_UVcuring) THEN
				uinDataAdress := DWORD_TO_UINT(RFID_Data.cRFID_UVcuring);
				uinDataAdress := uinDataAdress  MOD 16#100;							// only 0..255
				IF ((uinDataAdress >= 0) AND (uinDataAdress <= 255)) THEN
					SIf.Cur.stData.usiUVPinningLevel := 0;
					SIf.Cur.stData.usiUVPinningLevel.0 := SIf.Cur.abytData[uinDataAdress].0;
					SIf.Cur.stData.usiUVPinningLevel.1 := SIf.Cur.abytData[uinDataAdress].1;
					SIf.Cur.stData.usiUVPinningLevel.2 := SIf.Cur.abytData[uinDataAdress].2;
					SIf.Cur.stData.usiUVPinningLevel.3 := SIf.Cur.abytData[uinDataAdress].3;
		
					SIf.Cur.stData.usiUVLampLevel := 0;
					SIf.Cur.stData.usiUVLampLevel.0 := SIf.Cur.abytData[uinDataAdress].4;
					SIf.Cur.stData.usiUVLampLevel.1 := SIf.Cur.abytData[uinDataAdress].5;
					SIf.Cur.stData.usiUVLampLevel.2 := SIf.Cur.abytData[uinDataAdress].6;
					SIf.Cur.stData.usiUVLampLevel.3 := SIf.Cur.abytData[uinDataAdress].7;
				END_IF
			END_IF
			// Filename
			IF (dwoJobIntern = RFID_Data.cRFID_AllData) OR (dwoJobIntern = RFID_Data.cRFID_Filename) THEN
				uinDataAdress := DWORD_TO_UINT(RFID_Data.cRFID_Filename);
				uinDataLengh := DWORD_TO_UINT(SHR(RFID_Data.cRFID_Filename,16));
				uinDataAdress := uinDataAdress  MOD 16#100;							// only 0..255
				IF ((uinDataAdress >= 0) AND (uinDataAdress <= 255)) THEN
					strTemp := USINT_TO_STRING(SIf.Cur.abytData[uinDataAdress]);
					strTemp := TC2_STANDARD.CONCAT('-', strTemp);
					uliTemp := 0;
					uinDataAdress := uinDataAdress+1;	// Next signs
					Tc2_System.MEMCPY(destAddr := ADR(uliTemp), srcAddr := ADR(SIf.Cur.abytData[uinDataAdress]), n:= (uinDataLengh-1));
		
					SIf.Cur.stData.strFileName := TC2_STANDARD.CONCAT(ULINT_TO_STRING(uliTemp), strTemp);
				END_IF
			END_IF
			// Brush
			IF (dwoJobIntern = RFID_Data.cRFID_AllData) OR (dwoJobIntern = RFID_Data.cRFID_Brush) THEN
				uinDataAdress := DWORD_TO_UINT(RFID_Data.cRFID_Brush);
				uinDataAdress := uinDataAdress  MOD 16#100;							// only 0..255
				IF ((uinDataAdress >= 0) AND (uinDataAdress <= 255)) THEN
					SIf.Cur.stData.bolBrush := SIf.Cur.abytData[uinDataAdress].0;
					SIf.Cur.stData.bolBrushClean := SIf.Cur.abytData[uinDataAdress].1;
					SIf.Cur.stData.bolBrushFans := SIf.Cur.abytData[uinDataAdress].2;
					SIf.Cur.stData.bolGutterClean := SIf.Cur.abytData[uinDataAdress].6;
					SIf.Cur.stData.bolSpecialTray := SIf.Cur.abytData[uinDataAdress].7;
				END_IF
			END_IF
			
			// Tray ID
			IF (dwoJobIntern = RFID_Data.cRFID_TrayID) THEN
				uinDataAdress := DWORD_TO_UINT(RFID_Data.cRFID_TrayID);
				uinDataAdress := uinDataAdress  MOD 16#100;							// only 0..255
				IF ((uinDataAdress >= 0) AND (uinDataAdress <= 255)) THEN
					uinDataLengh := DWORD_TO_UINT(SHR(RFID_Data.cRFID_TrayID,16));
					SIf.Cur.stData.strTrayID := '';
					udiTemp := Tc2_System.MEMCPY(destAddr:=ADR(SIf.Cur.stData.strTrayID), srcAddr:=ADR(SIf.Cur.abytData[uinDataAdress]), n:=uinDataLengh);
				END_IF
			END_IF
	
			// Tag ID
			IF (dwoJobIntern = RFID_Data.cRFID_TagID) THEN
				uinDataAdress := DWORD_TO_UINT(RFID_Data.cRFID_TagID);
				uinDataAdress := uinDataAdress  MOD 16#100;							// only 0..255
				IF ((uinDataAdress >= 0) AND (uinDataAdress <= 255)) THEN
					uinDataLengh := DWORD_TO_UINT(SHR(RFID_Data.cRFID_TagID,16));
					SIf.Cur.stData.strTagID := '';
					udiTemp := Tc2_System.MEMCPY(destAddr:=ADR(SIf.Cur.stData.uliTagID), srcAddr:=ADR(pRFD_SIf^.stStatus.abyteUID), n:=8);
					SIf.Cur.stData.strTagID := FB_ULINT_TO_HEXSTRING(in_uliValue:= SIf.Cur.stData.uliTagID);	
				END_IF
			END_IF	
		//---------------------------------------
		//END_IF
			IF SIf.Cur.dwoJob = RFID_Data.cRFID_AllData THEN
				//IF udiTimeDelayRead >= 100 THEN // Wait 100ms
					IF dwoJobIntern = RFID_Data.cRFID_AllData THEN
						dwoJobIntern := RFID_Data.cRFID_TrayID;
						uinDataAdress := DWORD_TO_UINT(dwoJobIntern);
						uinDataAdress := uinDataAdress MOD 16#100;							// Maximum 255 data
						
						pRFD_SIf^.stCur.uinAdressData := uinDataAdress;
						pRFD_SIf^.stCur.uinAdressTag := DWORD_TO_UINT(dwoJobIntern);
						pRFD_SIf^.stCur.usiCount := DWORD_TO_USINT(SHR(dwoJobIntern,16));
				
						pRFD_SIf^.intCmd := RFD_Cmd.cRFD_CMD_Read;
						udiTimeDelayRead := 0;
					ELSIF dwoJobIntern = RFID_Data.cRFID_TrayID THEN
						dwoJobIntern := RFID_Data.cRFID_TagID;
						uinDataAdress := DWORD_TO_UINT(dwoJobIntern);
						uinDataAdress := uinDataAdress MOD 16#100;							// Maximum 255 data
						
						pRFD_SIf^.stCur.uinAdressData := uinDataAdress;
						pRFD_SIf^.stCur.uinAdressTag := DWORD_TO_UINT(dwoJobIntern);
						pRFD_SIf^.stCur.usiCount := DWORD_TO_USINT(SHR(dwoJobIntern,16));
				
						pRFD_SIf^.intCmd := RFD_Cmd.cRFD_CMD_MDS;
						udiTimeDelayRead := 0;
					ELSE
						bolAllFinished := TRUE;
					END_IF
				//ELSE
					udiTimeDelayRead := udiTimeDelayRead + me.FUBInfo.udiSample_ms;			
				//END_IF
			ELSE
				bolAllFinished := TRUE;
			END_IF
		END_IF
		// State Change Condition
		IF (pRFD_SIf^.stErr.bolErrorActive = TRUE) THEN  
			me.StateMachine.intStateNext :=  cSTA_ERROR;
		ELSIF (me.StateMachine.udiTimeInState_ms > SIf.Par.udiWriteTime_ms) THEN
			// SIf.Alm[4].strText := 'timeout wait on Data';
			pfbAlarmCtrl^.setAlarm(CIf.Info.intCtrlId,4,0,ADR(SIf.Alm),E_AlmState.RST,CIf.Job.eMe_ActivAlmClass);
			me.StateMachine.intStateNext :=  cSTA_ERROR;
		ELSIF (bolAllFinished = TRUE) THEN
			me.StateMachine.intStateNext := cSTA_READ;
		END_IF
	END_IF

	udiTimeDelayRead := udiTimeDelayRead + me.FUBInfo.udiSample_ms;



//--------------------------------------------------------------------------------------
// Exit action
	IF (me.StateMachine.intState<>me.StateMachine.intStateNext) THEN
		;
	END_IF
END_METHOD

METHOD PROTECTED sta_RUN : BOOL
// state implemetation
//--------------------------------------------------------------------------------------
// Entry action
	IF (me.StateMachine.intState<>me.StateMachine.intStateLastCycle) THEN
		me.StateMachine.intStateLastCycle := me.StateMachine.intState;
		bolNewTag := FALSE;
		me.SubStateMachine.intState := cRFW_SUB_WaitTag-1; // init first state - string
		me.SubStateMachine.intStateNext := cRFW_SUB_WaitTag;
		fbSimulationTimer.IN := FALSE;
		fbSimulationTimer.PT := UDINT_TO_TIME(SIf.Par.udiReadTime_ms / 2);
		fbSimulationTimer(); // set time/reset timer
		fbSimulationTimer.IN := TRUE; // start timer
		
	END_IF


//--------------------------------------------------------------------------------------
// Cyclic action
	IF (me.StateMachine.intState=me.StateMachine.intStateLastCycle) THEN

		// Simulation
		IF (CIf.SwCfg.bolSimulation) THEN
			fbSimulationTimer(); // simulation time
			IF (fbSimulationTimer.IN = FALSE) THEN
				fbSimulationTimer.IN := TRUE;
			END_IF
			IF pRFD_SIf^.intCmd <> RFD_Cmd.cRFD_CMD_DONE THEN
				pRFD_SIf^.intCmd := RFD_Cmd.cRFD_CMD_DONE;
			END_IF
			IF (fbSimulationTimer.Q) THEN
				fbSimulationTimer.IN := FALSE;
				IF SIf.Cur.bolPresent = FALSE THEN
					SIf.Cur.bolPresent := TRUE;
					SIf.Cur.stData.uliTagID := SIf.Cur.stData.uliTagID + 1;
					Tc2_System.MEMCPY(destAddr:=ADR(pRFD_SIf^.stStatus.abyteUID), srcAddr:=ADR(SIf.Cur.stData.uliTagID), n:=8);
				ELSE
					SIf.Cur.bolPresent := FALSE;
				END_IF
			END_IF
		END_IF
		
		// Function
		// If the RF ID Reader does not send automatically the Tag ID, read it if a new Tag is ready
		IF (SIf.Cfg.eTyp = E_Typ_RFW.RF310R) AND (CIf.SwCfg.bolSimulation = FALSE) THEN
			IF ((SIf.Cur.bolPresent = TRUE) AND (bolRENewTag = FALSE)) THEN
				bolNewTag := TRUE;
				bolRENewTag := TRUE;
			ELSIF (SIf.Cur.bolPresent = FALSE) THEN
				bolRENewTag := FALSE;
				bolNewTag := FALSE;
			END_IF
			
			//--------------------------------------------------------------------------------------
			// sub state machine for sequence
			CASE me.SubStateMachine.intState OF
				//--------------------------------------------------------------------------------------
				cRFW_SUB_WaitTag:
					IF (bolNewTag = TRUE) THEN
						me.SubStateMachine.intStateNext := cRFW_SUB_SendJob;
					END_IF
				
				cRFW_SUB_SendJob:
					pRFD_SIf^.stCur.uinAdressData :=0;
					pRFD_SIf^.stCur.uinAdressTag := DWORD_TO_UINT(RFID_Data.cRFID_TagID);
					pRFD_SIf^.stCur.usiCount := DWORD_TO_USINT(SHR(RFID_Data.cRFID_TagID,16));
				
					pRFD_SIf^.intCmd := RFD_Cmd.cRFD_CMD_MDS;
					
					me.SubStateMachine.intStateNext := cRFW_SUB_GetData;
					
				cRFW_SUB_GetData:
					IF pRFD_SIf^.intCmd = RFD_Cmd.cRFD_CMD_DONE THEN
						me.SubStateMachine.intStateNext := cRFW_SUB_CheckData;
					END_IF
				
				cRFW_SUB_CheckData:
					SIf.Cur.stData.strTagID := '';
					Tc2_System.MEMCPY(destAddr:=ADR(SIf.Cur.stData.uliTagID), srcAddr:=ADR(pRFD_SIf^.stStatus.abyteUID), n:=8);
					SIf.Cur.stData.strTagID := FB_ULINT_TO_HEXSTRING(in_uliValue:= SIf.Cur.stData.uliTagID);	

					IF (SIf.Cfg.bolGetTrayIDAuto = TRUE) THEN
						me.SubStateMachine.intStateNext := cRFW_SUB_SendJobTrayID;
					ELSE
						me.SubStateMachine.intStateNext := cRFW_SUB_Finished;
					END_IF
					
				cRFW_SUB_SendJobTrayID:
					uinDataAdress := DWORD_TO_UINT(RFID_Data.cRFID_TrayID);
					uinDataAdress := uinDataAdress MOD 16#100;							// Maximum 255 data
					uinDataLengh := DWORD_TO_UINT(SHR(RFID_Data.cRFID_TrayID,16));
					pRFD_SIf^.stCur.uinAdressData :=uinDataAdress;
					pRFD_SIf^.stCur.uinAdressTag := DWORD_TO_UINT(RFID_Data.cRFID_TrayID);
					pRFD_SIf^.stCur.usiCount := DWORD_TO_USINT(SHR(RFID_Data.cRFID_TrayID,16));
				
					pRFD_SIf^.intCmd := RFD_Cmd.cRFD_CMD_Read;
					
					me.SubStateMachine.intStateNext := cRFW_SUB_GetData;
					
				cRFW_SUB_GetDataTrayID:
					IF pRFD_SIf^.intCmd = RFD_Cmd.cRFD_CMD_DONE THEN
						me.SubStateMachine.intStateNext := cRFW_SUB_CheckData;
					END_IF
				
				cRFW_SUB_CheckDataTrayID:
					uinDataAdress := DWORD_TO_UINT(RFID_Data.cRFID_TrayID);
					uinDataAdress := uinDataAdress MOD 16#100;							// Maximum 255 data
					uinDataLengh := DWORD_TO_UINT(SHR(RFID_Data.cRFID_TrayID,16));
					SIf.Cur.stData.strTagID := '';
					Tc2_System.MEMCPY(destAddr:=ADR(SIf.Cur.stData.strTrayID), srcAddr:=ADR(pRFD_SIf^.stStatus.abyteUID[uinDataAdress]), n:=uinDataLengh);

					me.SubStateMachine.intStateNext := cRFW_SUB_Finished;
	
				cRFW_SUB_Finished:
					bolNewTag := FALSE;				
					me.SubStateMachine.intStateNext := cRFW_SUB_WaitTag;
					
			END_CASE
		ELSIF (SIf.Cfg.eTyp = E_Typ_RFW.RF382R) THEN
			SIf.Cur.stData.strTagID := '';
			Tc2_System.MEMCPY(destAddr:=ADR(SIf.Cur.stData.uliTagID), srcAddr:=ADR(pRFD_SIf^.stStatus.abyteUID), n:=8);
			SIf.Cur.stData.strTagID := FB_ULINT_TO_HEXSTRING(in_uliValue:= SIf.Cur.stData.uliTagID);	
			
		END_IF
		
		IF uliTagID_old <> SIf.Cur.stData.uliTagID THEN
			IF SIf.Cfg.bolDtChToLine_send = TRUE THEN
				IF SIf.Cfg.bolGetTrayIDAuto THEN
					intDtChnToLineState	:= fbDtChnToLine_NewRFID.Creat(In_uliTagID:= SIf.Cur.stData.uliTagID, In_strID:= SIf.Cur.stData.strTrayID);
				ELSE
					intDtChnToLineState	:= fbDtChnToLine_NewRFID.Creat(In_uliTagID:= SIf.Cur.stData.uliTagID, In_strID:= SIf.Cur.stData.strTagID);						
				END_IF
				IF intDtChnToLineState >= 0 THEN
					uliTagID_old := SIf.Cur.stData.uliTagID;
				ELSE
					// Set Alarm: SIf.Alm[6].strText := 'Data Channel Error Send Data';
					//pfbAlarmCtrl^.setAlarm(CIf.Info.intCtrlId,6,intDtChnToLineState,ADR(SIf.Alm),E_AlmState.RST,CIf.Job.eMe_ActivAlmClass);					
				END_IF
			ELSE
				uliTagID_old := SIf.Cur.stData.uliTagID;
			END_IF		
		END_IF
		
				
		// State Change Condition
		IF (pRFD_SIf^.stErr.bolErrorActive = TRUE) THEN  
			me.StateMachine.intStateNext :=  cSTA_ERROR;
		ELSIF ((me.intCmd=RFW_CmdState.cCMD_READ) OR (me.intCmd=RFW_CmdState.cCMD_WRITE)) AND (SIf.Cfg.eTyp = E_Typ_RFW.RF382R) THEN
			// SIf.Alm[5].strText := 'Command for this type of RFID not possible';
			pfbAlarmCtrl^.setAlarm(CIf.Info.intCtrlId,5,UDINT_TO_DINT(pRFD_SIf^.stErr.udiErrorID),ADR(SIf.Alm),E_AlmState.RST,CIf.Job.eMe_ActivAlmClass);			
		ELSIF (me.intCmd=RFW_CmdState.cCMD_READ) AND (me.SubStateMachine.intState = cRFW_SUB_WaitTag) THEN
			me.StateMachine.intStateNext := RFW_CmdState.cSTA_READBusy;
		ELSIF(me.intCmd=RFW_CmdState.cCMD_WRITE) AND (me.SubStateMachine.intState = cRFW_SUB_WaitTag) THEN
			me.StateMachine.intStateNext := RFW_CmdState.cSTA_WRITEBusy;
		ELSIF(me.intCmd=RFW_CmdState.cCMD_ON) THEN
			me.StateMachine.intStateNext := RFW_CmdState.cSTA_ONBusy;			
		END_IF
	END_IF




//--------------------------------------------------------------------------------------
// Exit action
	IF (me.StateMachine.intState<>me.StateMachine.intStateNext) THEN
		;		
	END_IF
END_METHOD

METHOD PROTECTED sta_RUNbusy : BOOL
// state implemetation
//--------------------------------------------------------------------------------------
// Entry action
	IF (me.StateMachine.intState<>me.StateMachine.intStateLastCycle) THEN
		me.StateMachine.intStateLastCycle := me.StateMachine.intState;
		bolNewTag := FALSE;
		me.SubStateMachine.intState := cRFW_SUB_WaitTag;
		SIf.Cur.dwoJob := RFID_Data.cRFID_TrayID;
		
		fbSimulationTimer.IN := FALSE;
		fbSimulationTimer.PT := UDINT_TO_TIME(SIf.Par.udiReadTime_ms / 2);
		fbSimulationTimer(); // set time/reset timer
		fbSimulationTimer.IN := TRUE; // start timer
		
	END_IF


//--------------------------------------------------------------------------------------
// Cyclic action
	IF (me.StateMachine.intState=me.StateMachine.intStateLastCycle) THEN

		// Simulation
		IF (CIf.SwCfg.bolSimulation) THEN
			fbSimulationTimer(); // simulation time
			IF (fbSimulationTimer.Q) THEN
				;
			END_IF
		END_IF
		
		// Function
		
		// State Change Condition
		IF (pRFD_SIf^.stErr.bolErrorActive = TRUE) THEN  
			me.StateMachine.intStateNext :=  cSTA_ERROR;
		ELSIF(me.intCmd=cCMD_READ) THEN
			me.StateMachine.intStateNext := cSTA_READBusy;
		ELSIF(me.intCmd=cCMD_WRITE) THEN
			me.StateMachine.intStateNext := cSTA_WRITEBusy;
		ELSE
			me.StateMachine.intStateNext := cSTA_RUN;
		END_IF
	END_IF




//--------------------------------------------------------------------------------------
// Exit action
	IF (me.StateMachine.intState<>me.StateMachine.intStateNext) THEN
		;		
	END_IF
END_METHOD

METHOD PROTECTED sta_WRITE : BOOL
// state implemetation
//--------------------------------------------------------------------------------------
// Entry action
	IF (me.StateMachine.intState<>me.StateMachine.intStateLastCycle) THEN
		me.StateMachine.intStateLastCycle := me.StateMachine.intState;

	END_IF


//--------------------------------------------------------------------------------------
// Cyclic action
	IF (me.StateMachine.intState=me.StateMachine.intStateLastCycle) THEN

		// Simulation
		IF (CIf.SwCfg.bolSimulation) THEN
			;
		END_IF
		
		// State Change Condition
		IF(me.intCmd=cCMD_RUN) THEN
			me.StateMachine.intStateNext := cSTA_RUNBusy;
		ELSIF(me.intCmd=RFW_CmdState.cCMD_READ) THEN
			me.StateMachine.intStateNext := RFW_CmdState.cSTA_READBusy;
		ELSIF ((me.intCmd=RFW_CmdState.cCMD_READ) OR (me.intCmd=RFW_CmdState.cCMD_WRITE)) AND (SIf.Cfg.eTyp = E_Typ_RFW.RF382R) THEN
			// SIf.Alm[5].strText := 'Command for this type of RFID not possible';
			pfbAlarmCtrl^.setAlarm(CIf.Info.intCtrlId,5,UDINT_TO_DINT(pRFD_SIf^.stErr.udiErrorID),ADR(SIf.Alm),E_AlmState.RST,CIf.Job.eMe_ActivAlmClass);	
		ELSIF(me.intCmd=RFW_CmdState.cCMD_WRITE) THEN
			me.StateMachine.intStateNext := RFW_CmdState.cSTA_WRITEBusy;
		ELSIF(me.intCmd=RFW_CmdState.cCMD_ON) THEN
			me.StateMachine.intStateNext := RFW_CmdState.cSTA_ONBusy;			
		END_IF
	END_IF




//--------------------------------------------------------------------------------------
// Exit action
	IF (me.StateMachine.intState<>me.StateMachine.intStateNext) THEN
		;
	END_IF
END_METHOD

METHOD PROTECTED sta_WRITEBusy : BOOL
// state implemetation
//--------------------------------------------------------------------------------------
// Entry action
	IF (me.StateMachine.intState<>me.StateMachine.intStateLastCycle) THEN
		me.StateMachine.intStateLastCycle := me.StateMachine.intState;

		fbSimulationTimer.IN := FALSE;
		fbSimulationTimer.PT := UDINT_TO_TIME(SIf.Par.udiWriteTime_ms / 2);
		fbSimulationTimer(); // set time/reset timer
		fbSimulationTimer.IN := TRUE; // start timer
		
		IF SIf.Cur.dwoJob = 0 THEN
			SIf.Cur.dwoJob := RFID_Data.cRFID_AllData;
		END_IF
		
